LIN {X 0,Y 625.989,Z 663.19,A -85,B 0,C 180,E1 6456.402,E2 6456.402} C_VEL
LIN {X 0,Y 626.113,Z 663.19,A -85,B 0,C 180,E1 6463.797,E2 6463.797} C_VEL
LIN {X 0,Y 626.332,Z 663.19,A -85,B 0,C 180,E1 6470.922,E2 6470.922} C_VEL
LIN {X 0,Y 626.466,Z 663.19,A -85,B 0,C 180,E1 6477.902,E2 6477.902} C_VEL
LIN {X 0,Y 626.549,Z 663.19,A -85,B 0,C 180,E1 6484.849,E2 6484.849} C_VEL
LIN {X 0,Y 626.308,Z 663.19,A -85,B 0,C 180,E1 6493.295,E2 6493.295} C_VEL
LIN {X 0,Y 626.36,Z 663.19,A -85,B 0,C 180,E1 6501.237,E2 6501.237} C_VEL
LIN {X 0,Y 626.317,Z 663.19,A -85,B 0,C 180,E1 6509.77,E2 6509.77} C_VEL
LIN {X 0,Y 626.419,Z 663.19,A -85,B 0,C 180,E1 6518.14,E2 6518.14} C_VEL
LIN {X 0,Y 626.399,Z 664.346,A -85,B 0,C 180,E1 6525.792,E2 6525.792} C_VEL
LIN {X 0,Y 651.869,Z 715.355,A -85,B 0,C 180,E1 6528.472,E2 6528.472} C_VEL
LIN {X 0,Y 648.177,Z 791.571,A -85,B 0,C 180,E1 6530.446,E2 6530.446} C_VEL
LIN {X 0,Y 642.47,Z 861.614,A -85,B 0,C 180,E1 6533.738,E2 6533.738} C_VEL
LIN {X 0,Y 636.508,Z 924.999,A -85,B 0,C 180,E1 6538.337,E2 6538.337} C_VEL
LIN {X 0,Y 631.672,Z 978.511,A -85,B 0,C 180,E1 6544.011,E2 6544.011} C_VEL
LIN {X 0,Y 628.979,Z 1020.004,A -85,B 0,C 180,E1 6550.536,E2 6550.536} C_VEL
LIN {X 0,Y 627.568,Z 1047.097,A -85,B 0,C 180,E1 6557.439,E2 6557.439} C_VEL
LIN {X 0,Y 626.974,Z 1058.972,A -85,B 0,C 180,E1 6563.751,E2 6563.751} C_VEL
LIN {X 0,Y 627.176,Z 1059.603,A -85,B 0,C 180,E1 6569.307,E2 6569.307} C_VEL
LIN {X 0,Y 627.134,Z 1049.647,A -85,B 0,C 180,E1 6575.55,E2 6575.55} C_VEL
LIN {X 0,Y 627.887,Z 1027.464,A -85,B 0,C 180,E1 6581.846,E2 6581.846} C_VEL
LIN {X 0,Y 629.7,Z 1006.621,A -85,B 0,C 180,E1 6585.788,E2 6585.788} C_VEL
LIN {X 0,Y 622.562,Z 990.323,A -85,B 0,C 180,E1 6588.601,E2 6588.601} C_VEL
LIN {X 0,Y 627.357,Z 940.981,A -85,B 0,C 180,E1 6594.452,E2 6594.452} C_VEL
LIN {X 0,Y 633.854,Z 879.366,A -85,B 0,C 180,E1 6599.458,E2 6599.458} C_VEL
LIN {X 0,Y 640.199,Z 811.845,A -85,B 0,C 180,E1 6603.087,E2 6603.087} C_VEL
LIN {X 0,Y 644.763,Z 741.705,A -85,B 0,C 180,E1 6605.351,E2 6605.351} C_VEL
LIN {X 0,Y 644.279,Z 712.829,A -85,B 0,C 180,E1 6606.02,E2 6606.02} C_VEL
LIN {X 0,Y 618.028,Z 663.19,A -85,B 0,C 180,E1 6608.956,E2 6608.956} C_VEL
LIN {X 0,Y 618.105,Z 663.19,A -85,B 0,C 180,E1 6617.545,E2 6617.545} C_VEL
LIN {X 0,Y 618.102,Z 663.19,A -85,B 0,C 180,E1 6626.48,E2 6626.48} C_VEL
LIN {X 0,Y 618.278,Z 663.19,A -85,B 0,C 180,E1 6634.575,E2 6634.575} C_VEL
LIN {X 0,Y 618.593,Z 663.19,A -85,B 0,C 180,E1 6643.626,E2 6643.626} C_VEL
LIN {X 0,Y 618.803,Z 663.19,A -85,B 0,C 180,E1 6650.842,E2 6650.842} C_VEL
LIN {X 0,Y 619.166,Z 663.19,A -85,B 0,C 180,E1 6657.908,E2 6657.908} C_VEL
LIN {X 0,Y 618.585,Z 663.19,A -85,B 0,C 180,E1 6666.87,E2 6666.87} C_VEL
LIN {X 0,Y 618.331,Z 663.19,A -85,B 0,C 180,E1 6674.952,E2 6674.952} C_VEL
LIN {X 0,Y 618.059,Z 663.19,A -85,B 0,C 180,E1 6683.065,E2 6683.065} C_VEL
LIN {X 0,Y 618.548,Z 663.19,A -85,B 0,C 180,E1 6691.859,E2 6691.859} C_VEL
LIN {X 0,Y 618.263,Z 663.19,A -85,B 0,C 180,E1 6700.603,E2 6700.603} C_VEL
LIN {X 0,Y 618.318,Z 665.155,A -85,B 0,C 180,E1 6708.054,E2 6708.054} C_VEL
LIN {X 0,Y 645.805,Z 718.768,A -85,B 0,C 180,E1 6710.981,E2 6710.981} C_VEL
LIN {X 0,Y 642.302,Z 793.069,A -85,B 0,C 180,E1 6712.772,E2 6712.772} C_VEL
LIN {X 0,Y 636.489,Z 863.014,A -85,B 0,C 180,E1 6715.883,E2 6715.883} C_VEL
LIN {X 0,Y 630.05,Z 926.753,A -85,B 0,C 180,E1 6720.294,E2 6720.294} C_VEL
LIN {X 0,Y 624.493,Z 981.34,A -85,B 0,C 180,E1 6725.846,E2 6725.846} C_VEL
LIN {X 0,Y 621.095,Z 1024.089,A -85,B 0,C 180,E1 6732.231,E2 6732.231} C_VEL
LIN {X 0,Y 619.771,Z 1052.761,A -85,B 0,C 180,E1 6738.919,E2 6738.919} C_VEL
LIN {X 0,Y 619.545,Z 1067.017,A -85,B 0,C 180,E1 6745.086,E2 6745.086} C_VEL
LIN {X 0,Y 619.231,Z 1069.804,A -85,B 0,C 180,E1 6752.105,E2 6752.105} C_VEL
LIN {X 0,Y 619.104,Z 1060.28,A -85,B 0,C 180,E1 6758.451,E2 6758.451} C_VEL
LIN {X 0,Y 619.864,Z 1039.304,A -85,B 0,C 180,E1 6764.658,E2 6764.658} C_VEL
LIN {X 0,Y 622.106,Z 1006.633,A -85,B 0,C 180,E1 6770.698,E2 6770.698} C_VEL
LIN {X 0,Y 626.721,Z 958.006,A -85,B 0,C 180,E1 6776.784,E2 6776.784} C_VEL
LIN {X 0,Y 632.897,Z 898.514,A -85,B 0,C 180,E1 6781.89,E2 6781.89} C_VEL
LIN {X 0,Y 639.339,Z 831.694,A -85,B 0,C 180,E1 6785.706,E2 6785.706} C_VEL
LIN {X 0,Y 644.355,Z 760.024,A -85,B 0,C 180,E1 6788.194,E2 6788.194} C_VEL
LIN {X 0,Y 644.727,Z 712.454,A -85,B 0,C 180,E1 6789.202,E2 6789.202} C_VEL
LIN {X 0,Y 617.986,Z 663.19,A -85,B 0,C 180,E1 6792.181,E2 6792.181} C_VEL
LIN {X 0,Y 617.872,Z 663.19,A -85,B 0,C 180,E1 6801.195,E2 6801.195} C_VEL
LIN {X 0,Y 618.195,Z 663.19,A -85,B 0,C 180,E1 6809.763,E2 6809.763} C_VEL
LIN {X 0,Y 618.409,Z 663.19,A -85,B 0,C 180,E1 6819.136,E2 6819.136} C_VEL
LIN {X 0,Y 618.785,Z 663.19,A -85,B 0,C 180,E1 6827.95,E2 6827.95} C_VEL
LIN {X 0,Y 618.905,Z 663.19,A -85,B 0,C 180,E1 6836.47,E2 6836.47} C_VEL
LIN {X 0,Y 618.526,Z 663.19,A -85,B 0,C 180,E1 6844.912,E2 6844.912} C_VEL
LIN {X 0,Y 618.606,Z 663.19,A -85,B 0,C 180,E1 6852.022,E2 6852.022} C_VEL
LIN {X 0,Y 618.434,Z 663.19,A -85,B 0,C 180,E1 6860.83,E2 6860.83} C_VEL
LIN {X 0,Y 618.309,Z 663.19,A -85,B 0,C 180,E1 6869.466,E2 6869.466} C_VEL
LIN {X 0,Y 618.325,Z 663.19,A -85,B 0,C 180,E1 6877.15,E2 6877.15} C_VEL
LIN {X 0,Y 618.439,Z 665.18,A -85,B 0,C 180,E1 6885.154,E2 6885.154} C_VEL
LIN {X 0,Y 645.566,Z 717.694,A -85,B 0,C 180,E1 6888.064,E2 6888.064} C_VEL
LIN {X 0,Y 641.566,Z 793.048,A -85,B 0,C 180,E1 6890.072,E2 6890.072} C_VEL
LIN {X 0,Y 635.518,Z 862.685,A -85,B 0,C 180,E1 6893.399,E2 6893.399} C_VEL
LIN {X 0,Y 629.093,Z 926.353,A -85,B 0,C 180,E1 6898.095,E2 6898.095} C_VEL
LIN {X 0,Y 623.955,Z 979.19,A -85,B 0,C 180,E1 6903.799,E2 6903.799} C_VEL
LIN {X 0,Y 621.072,Z 1020.648,A -85,B 0,C 180,E1 6910.454,E2 6910.454} C_VEL
LIN {X 0,Y 619.649,Z 1046.987,A -85,B 0,C 180,E1 6917.276,E2 6917.276} C_VEL
LIN {X 0,Y 618.987,Z 1058.942,A -85,B 0,C 180,E1 6923.67,E2 6923.67} C_VEL
LIN {X 0,Y 619.176,Z 1059.632,A -85,B 0,C 180,E1 6929.298,E2 6929.298} C_VEL
LIN {X 0,Y 619.146,Z 1049.756,A -85,B 0,C 180,E1 6935.622,E2 6935.622} C_VEL
LIN {X 0,Y 619.919,Z 1029.339,A -85,B 0,C 180,E1 6941.604,E2 6941.604} C_VEL
LIN {X 0,Y 622.168,Z 996.079,A -85,B 0,C 180,E1 6947.738,E2 6947.738} C_VEL
LIN {X 0,Y 622.562,Z 990.323,A -85,B 0,C 180,E1 6948.601,E2 6948.601} C_VEL
LIN {X 0,Y 617.22,Z 971.758,A -85,B 0,C 180,E1 6951.357,E2 6951.357} C_VEL
LIN {X 0,Y 622.951,Z 916.676,A -85,B 0,C 180,E1 6957.041,E2 6957.041} C_VEL
LIN {X 0,Y 629.604,Z 853.137,A -85,B 0,C 180,E1 6961.489,E2 6961.489} C_VEL
LIN {X 0,Y 635.961,Z 781.489,A -85,B 0,C 180,E1 6964.683,E2 6964.683} C_VEL
LIN {X 0,Y 638.105,Z 715.966,A -85,B 0,C 180,E1 6966.419,E2 6966.419} C_VEL
LIN {X 0,Y 609.903,Z 663.19,A -85,B 0,C 180,E1 6969.693,E2 6969.693} C_VEL
LIN {X 0,Y 610.126,Z 663.19,A -85,B 0,C 180,E1 6977.154,E2 6977.154} C_VEL
LIN {X 0,Y 610.092,Z 663.19,A -85,B 0,C 180,E1 6986.372,E2 6986.372} C_VEL
LIN {X 0,Y 610.278,Z 663.19,A -85,B 0,C 180,E1 6995.086,E2 6995.086} C_VEL
LIN {X 0,Y 610.527,Z 663.19,A -85,B 0,C 180,E1 7003.404,E2 7003.404} C_VEL
LIN {X 0,Y 610.82,Z 663.19,A -85,B 0,C 180,E1 7010.721,E2 7010.721} C_VEL
LIN {X 0,Y 611.183,Z 663.19,A -85,B 0,C 180,E1 7017.881,E2 7017.881} C_VEL
LIN {X 0,Y 610.717,Z 663.19,A -85,B 0,C 180,E1 7026.437,E2 7026.437} C_VEL
LIN {X 0,Y 610.275,Z 663.19,A -85,B 0,C 180,E1 7035.154,E2 7035.154} C_VEL
LIN {X 0,Y 610.13,Z 663.19,A -85,B 0,C 180,E1 7042.697,E2 7042.697} C_VEL
LIN {X 0,Y 610.501,Z 663.19,A -85,B 0,C 180,E1 7051.026,E2 7051.026} C_VEL
LIN {X 0,Y 610.256,Z 663.19,A -85,B 0,C 180,E1 7059.382,E2 7059.382} C_VEL
LIN {X 0,Y 610.188,Z 664.755,A -85,B 0,C 180,E1 7067.37,E2 7067.37} C_VEL
LIN {X 0,Y 639.531,Z 721.3,A -85,B 0,C 180,E1 7070.569,E2 7070.569} C_VEL
LIN {X 0,Y 635.739,Z 794.861,A -85,B 0,C 180,E1 7072.394,E2 7072.394} C_VEL
LIN {X 0,Y 629.598,Z 864.163,A -85,B 0,C 180,E1 7075.528,E2 7075.528} C_VEL
LIN {X 0,Y 622.672,Z 928.343,A -85,B 0,C 180,E1 7080.05,E2 7080.05} C_VEL
LIN {X 0,Y 616.761,Z 982.879,A -85,B 0,C 180,E1 7085.726,E2 7085.726} C_VEL
LIN {X 0,Y 613.197,Z 1025.473,A -85,B 0,C 180,E1 7092.258,E2 7092.258} C_VEL
LIN {X 0,Y 611.857,Z 1054.394,A -85,B 0,C 180,E1 7099.288,E2 7099.288} C_VEL
LIN {X 0,Y 611.057,Z 1068.735,A -85,B 0,C 180,E1 7106.443,E2 7106.443} C_VEL
LIN {X 0,Y 611.217,Z 1069.804,A -85,B 0,C 180,E1 7112.133,E2 7112.133} C_VEL
LIN {X 0,Y 611.106,Z 1060.28,A -85,B 0,C 180,E1 7118.563,E2 7118.563} C_VEL
LIN {X 0,Y 611.921,Z 1039.774,A -85,B 0,C 180,E1 7124.74,E2 7124.74} C_VEL
LIN {X 0,Y 614.345,Z 1006.631,A -85,B 0,C 180,E1 7130.972,E2 7130.972} C_VEL
LIN {X 0,Y 619.276,Z 958.172,A -85,B 0,C 180,E1 7137.113,E2 7137.113} C_VEL
LIN {X 0,Y 625.962,Z 898.034,A -85,B 0,C 180,E1 7142.322,E2 7142.322} C_VEL
LIN {X 0,Y 632.78,Z 831.525,A -85,B 0,C 180,E1 7146.141,E2 7146.141} C_VEL
LIN {X 0,Y 638.057,Z 759.411,A -85,B 0,C 180,E1 7148.655,E2 7148.655} C_VEL
LIN {X 0,Y 638.305,Z 715.18,A -85,B 0,C 180,E1 7149.625,E2 7149.625} C_VEL
LIN {X 0,Y 610.038,Z 663.19,A -85,B 0,C 180,E1 7152.757,E2 7152.757} C_VEL
LIN {X 0,Y 609.871,Z 663.19,A -85,B 0,C 180,E1 7161.558,E2 7161.558} C_VEL
LIN {X 0,Y 610.255,Z 663.19,A -85,B 0,C 180,E1 7170.97,E2 7170.97} C_VEL
LIN {X 0,Y 610.396,Z 663.19,A -85,B 0,C 180,E1 7180.369,E2 7180.369} C_VEL
LIN {X 0,Y 610.575,Z 663.19,A -85,B 0,C 180,E1 7189.239,E2 7189.239} C_VEL
LIN {X 0,Y 610.917,Z 663.19,A -85,B 0,C 180,E1 7196.424,E2 7196.424} C_VEL
LIN {X 0,Y 611.171,Z 663.19,A -85,B 0,C 180,E1 7203.544,E2 7203.544} C_VEL
LIN {X 0,Y 610.553,Z 663.19,A -85,B 0,C 180,E1 7212.183,E2 7212.183} C_VEL
LIN {X 0,Y 610.375,Z 663.19,A -85,B 0,C 180,E1 7221.118,E2 7221.118} C_VEL
LIN {X 0,Y 610.299,Z 663.19,A -85,B 0,C 180,E1 7228.992,E2 7228.992} C_VEL
LIN {X 0,Y 610.296,Z 663.19,A -85,B 0,C 180,E1 7237.52,E2 7237.52} C_VEL
LIN {X 0,Y 610.298,Z 665.046,A -85,B 0,C 180,E1 7244.451,E2 7244.451} C_VEL
LIN {X 0,Y 639.271,Z 719.493,A -85,B 0,C 180,E1 7247.644,E2 7247.644} C_VEL
LIN {X 0,Y 634.992,Z 794.438,A -85,B 0,C 180,E1 7249.684,E2 7249.684} C_VEL
LIN {X 0,Y 628.464,Z 864.635,A -85,B 0,C 180,E1 7253.103,E2 7253.103} C_VEL
LIN {X 0,Y 621.74,Z 927.168,A -85,B 0,C 180,E1 7257.798,E2 7257.798} C_VEL
LIN {X 0,Y 616.267,Z 979.509,A -85,B 0,C 180,E1 7263.535,E2 7263.535} C_VEL
LIN {X 0,Y 613.144,Z 1020.442,A -85,B 0,C 180,E1 7270.191,E2 7270.191} C_VEL
LIN {X 0,Y 611.714,Z 1046.878,A -85,B 0,C 180,E1 7277.108,E2 7277.108} C_VEL
LIN {X 0,Y 611.011,Z 1058.913,A -85,B 0,C 180,E1 7283.587,E2 7283.587} C_VEL
LIN {X 0,Y 611.197,Z 1059.66,A -85,B 0,C 180,E1 7289.289,E2 7289.289} C_VEL
LIN {X 0,Y 611.148,Z 1049.864,A -85,B 0,C 180,E1 7295.696,E2 7295.696} C_VEL
LIN {X 0,Y 611.978,Z 1029.194,A -85,B 0,C 180,E1 7301.832,E2 7301.832} C_VEL
LIN {X 0,Y 614.41,Z 995.857,A -85,B 0,C 180,E1 7308.047,E2 7308.047} C_VEL
LIN {X 0,Y 617.22,Z 971.758,A -85,B 0,C 180,E1 7311.357,E2 7311.357} C_VEL
LIN {X 0,Y 611.43,Z 951.715,A -85,B 0,C 180,E1 7314.042,E2 7314.042} C_VEL
LIN {X 0,Y 618.594,Z 892.06,A -85,B 0,C 180,E1 7319.381,E2 7319.381} C_VEL
LIN {X 0,Y 625.879,Z 825.182,A -85,B 0,C 180,E1 7323.375,E2 7323.375} C_VEL
LIN {X 0,Y 631.561,Z 752.877,A -85,B 0,C 180,E1 7325.996,E2 7325.996} C_VEL
LIN {X 0,Y 631.694,Z 718.464,A -85,B 0,C 180,E1 7326.856,E2 7326.856} C_VEL
LIN {X 0,Y 601.853,Z 663.19,A -85,B 0,C 180,E1 7330.342,E2 7330.342} C_VEL
LIN {X 0,Y 602,Z 663.19,A -85,B 0,C 180,E1 7338.098,E2 7338.098} C_VEL
LIN {X 0,Y 602.138,Z 663.19,A -85,B 0,C 180,E1 7347.203,E2 7347.203} C_VEL
LIN {X 0,Y 602.32,Z 663.19,A -85,B 0,C 180,E1 7355.449,E2 7355.449} C_VEL
LIN {X 0,Y 602.823,Z 663.19,A -85,B 0,C 180,E1 7364.687,E2 7364.687} C_VEL
LIN {X 0,Y 602.465,Z 663.19,A -85,B 0,C 180,E1 7372.051,E2 7372.051} C_VEL
LIN {X 0,Y 602.554,Z 663.19,A -85,B 0,C 180,E1 7379.294,E2 7379.294} C_VEL
LIN {X 0,Y 602.709,Z 663.19,A -85,B 0,C 180,E1 7386.523,E2 7386.523} C_VEL
LIN {X 0,Y 602.233,Z 663.19,A -85,B 0,C 180,E1 7395.361,E2 7395.361} C_VEL
LIN {X 0,Y 602.022,Z 663.19,A -85,B 0,C 180,E1 7403.164,E2 7403.164} C_VEL
LIN {X 0,Y 602.505,Z 663.19,A -85,B 0,C 180,E1 7411.111,E2 7411.111} C_VEL
LIN {X 0,Y 602.233,Z 663.19,A -85,B 0,C 180,E1 7420.011,E2 7420.011} C_VEL
LIN {X 0,Y 602.125,Z 664.619,A -85,B 0,C 180,E1 7426.675,E2 7426.675} C_VEL
LIN {X 0,Y 633.316,Z 722.987,A -85,B 0,C 180,E1 7430.135,E2 7430.135} C_VEL
LIN {X 0,Y 629.168,Z 797.343,A -85,B 0,C 180,E1 7432.031,E2 7432.031} C_VEL
LIN {X 0,Y 622.501,Z 867.6,A -85,B 0,C 180,E1 7435.297,E2 7435.297} C_VEL
LIN {X 0,Y 615.215,Z 930.645,A -85,B 0,C 180,E1 7439.873,E2 7439.873} C_VEL
LIN {X 0,Y 608.925,Z 985.452,A -85,B 0,C 180,E1 7445.739,E2 7445.739} C_VEL
LIN {X 0,Y 605.274,Z 1026.854,A -85,B 0,C 180,E1 7452.285,E2 7452.285} C_VEL
LIN {X 0,Y 603.907,Z 1055.519,A -85,B 0,C 180,E1 7459.511,E2 7459.511} C_VEL
LIN {X 0,Y 603.066,Z 1068.735,A -85,B 0,C 180,E1 7466.396,E2 7466.396} C_VEL
LIN {X 0,Y 603.205,Z 1069.805,A -85,B 0,C 180,E1 7472.161,E2 7472.161} C_VEL
LIN {X 0,Y 603.127,Z 1060.281,A -85,B 0,C 180,E1 7478.677,E2 7478.677} C_VEL
LIN {X 0,Y 603.972,Z 1040.223,A -85,B 0,C 180,E1 7484.829,E2 7484.829} C_VEL
LIN {X 0,Y 606.511,Z 1007.671,A -85,B 0,C 180,E1 7491.09,E2 7491.09} C_VEL
LIN {X 0,Y 611.714,Z 959.739,A -85,B 0,C 180,E1 7497.298,E2 7497.298} C_VEL
LIN {X 0,Y 618.824,Z 899.5,A -85,B 0,C 180,E1 7502.624,E2 7502.624} C_VEL
LIN {X 0,Y 626.099,Z 832.698,A -85,B 0,C 180,E1 7506.525,E2 7506.525} C_VEL
LIN {X 0,Y 631.688,Z 760.974,A -85,B 0,C 180,E1 7509.072,E2 7509.072} C_VEL
LIN {X 0,Y 632.081,Z 718.258,A -85,B 0,C 180,E1 7510.039,E2 7510.039} C_VEL
LIN {X 0,Y 602.03,Z 663.19,A -85,B 0,C 180,E1 7513.5,E2 7513.5} C_VEL
LIN {X 0,Y 601.938,Z 663.19,A -85,B 0,C 180,E1 7522.519,E2 7522.519} C_VEL
LIN {X 0,Y 602.161,Z 663.19,A -85,B 0,C 180,E1 7530.542,E2 7530.542} C_VEL
LIN {X 0,Y 602.36,Z 663.19,A -85,B 0,C 180,E1 7540.097,E2 7540.097} C_VEL
LIN {X 0,Y 602.585,Z 663.19,A -85,B 0,C 180,E1 7549.095,E2 7549.095} C_VEL
LIN {X 0,Y 602.92,Z 663.19,A -85,B 0,C 180,E1 7556.376,E2 7556.376} C_VEL
LIN {X 0,Y 603.132,Z 663.19,A -85,B 0,C 180,E1 7563.591,E2 7563.591} C_VEL
LIN {X 0,Y 602.496,Z 663.19,A -85,B 0,C 180,E1 7572.348,E2 7572.348} C_VEL
LIN {X 0,Y 602.345,Z 663.19,A -85,B 0,C 180,E1 7581.414,E2 7581.414} C_VEL
LIN {X 0,Y 602.251,Z 663.19,A -85,B 0,C 180,E1 7589.694,E2 7589.694} C_VEL
LIN {X 0,Y 602.283,Z 663.19,A -85,B 0,C 180,E1 7598.108,E2 7598.108} C_VEL
LIN {X 0,Y 602.263,Z 665.134,A -85,B 0,C 180,E1 7603.728,E2 7603.728} C_VEL
LIN {X 0,Y 632.957,Z 722.137,A -85,B 0,C 180,E1 7607.233,E2 7607.233} C_VEL
LIN {X 0,Y 628.153,Z 798.434,A -85,B 0,C 180,E1 7609.384,E2 7609.384} C_VEL
LIN {X 0,Y 621.227,Z 868.652,A -85,B 0,C 180,E1 7612.93,E2 7612.93} C_VEL
LIN {X 0,Y 614.205,Z 930.063,A -85,B 0,C 180,E1 7617.685,E2 7617.685} C_VEL
LIN {X 0,Y 608.374,Z 982.733,A -85,B 0,C 180,E1 7623.67,E2 7623.67} C_VEL
LIN {X 0,Y 605.22,Z 1021.68,A -85,B 0,C 180,E1 7630.229,E2 7630.229} C_VEL
LIN {X 0,Y 603.785,Z 1046.768,A -85,B 0,C 180,E1 7636.936,E2 7636.936} C_VEL
LIN {X 0,Y 602.999,Z 1059.027,A -85,B 0,C 180,E1 7643.702,E2 7643.702} C_VEL
LIN {X 0,Y 603.196,Z 1059.689,A -85,B 0,C 180,E1 7649.279,E2 7649.279} C_VEL
LIN {X 0,Y 603.162,Z 1050.094,A -85,B 0,C 180,E1 7655.718,E2 7655.718} C_VEL
LIN {X 0,Y 604.04,Z 1029.061,A -85,B 0,C 180,E1 7662.065,E2 7662.065} C_VEL
LIN {X 0,Y 606.693,Z 995.443,A -85,B 0,C 180,E1 7668.394,E2 7668.394} C_VEL
LIN {X 0,Y 611.43,Z 951.715,A -85,B 0,C 180,E1 7674.042,E2 7674.042} C_VEL
LIN {X 0,Y 606.879,Z 929.837,A -85,B 0,C 180,E1 7676.636,E2 7676.636} C_VEL
LIN {X 0,Y 614.715,Z 866.262,A -85,B 0,C 180,E1 7681.561,E2 7681.561} C_VEL
LIN {X 0,Y 621.985,Z 797.253,A -85,B 0,C 180,E1 7685.021,E2 7685.021} C_VEL
LIN {X 0,Y 626.889,Z 727.794,A -85,B 0,C 180,E1 7687.011,E2 7687.011} C_VEL
LIN {X 0,Y 602.756,Z 679.837,A -85,B 0,C 180,E1 7689.849,E2 7689.849} C_VEL
LIN {X 0,Y 593.856,Z 663.19,A -85,B 0,C 180,E1 7691.089,E2 7691.089} C_VEL
LIN {X 0,Y 593.937,Z 663.19,A -85,B 0,C 180,E1 7699.355,E2 7699.355} C_VEL
LIN {X 0,Y 594.246,Z 663.19,A -85,B 0,C 180,E1 7708.744,E2 7708.744} C_VEL
LIN {X 0,Y 594.424,Z 663.19,A -85,B 0,C 180,E1 7718.287,E2 7718.287} C_VEL
LIN {X 0,Y 595.208,Z 663.19,A -85,B 0,C 180,E1 7727.498,E2 7727.498} C_VEL
LIN {X 0,Y 595.176,Z 663.19,A -85,B 0,C 180,E1 7737.824,E2 7737.824} C_VEL
LIN {X 0,Y 594.672,Z 663.19,A -85,B 0,C 180,E1 7746.611,E2 7746.611} C_VEL
LIN {X 0,Y 594.189,Z 663.19,A -85,B 0,C 180,E1 7755.574,E2 7755.574} C_VEL
LIN {X 0,Y 593.997,Z 663.19,A -85,B 0,C 180,E1 7763.349,E2 7763.349} C_VEL
LIN {X 0,Y 594.505,Z 663.19,A -85,B 0,C 180,E1 7771.577,E2 7771.577} C_VEL
LIN {X 0,Y 594.145,Z 663.19,A -85,B 0,C 180,E1 7780.669,E2 7780.669} C_VEL
LIN {X 0,Y 594.206,Z 665.179,A -85,B 0,C 180,E1 7785.982,E2 7785.982} C_VEL
LIN {X 0,Y 627.136,Z 724.807,A -85,B 0,C 180,E1 7789.696,E2 7789.696} C_VEL
LIN {X 0,Y 622.711,Z 798.447,A -85,B 0,C 180,E1 7791.613,E2 7791.613} C_VEL
LIN {X 0,Y 615.771,Z 867.404,A -85,B 0,C 180,E1 7794.855,E2 7794.855} C_VEL
LIN {X 0,Y 607.996,Z 930.747,A -85,B 0,C 180,E1 7799.488,E2 7799.488} C_VEL
LIN {X 0,Y 601.331,Z 985.45,A -85,B 0,C 180,E1 7805.412,E2 7805.412} C_VEL
LIN {X 0,Y 597.417,Z 1026.619,A -85,B 0,C 180,E1 7811.999,E2 7811.999} C_VEL
LIN {X 0,Y 595.916,Z 1055.519,A -85,B 0,C 180,E1 7819.369,E2 7819.369} C_VEL
LIN {X 0,Y 595.075,Z 1068.735,A -85,B 0,C 180,E1 7826.348,E2 7826.348} C_VEL
LIN {X 0,Y 595.196,Z 1069.805,A -85,B 0,C 180,E1 7832.191,E2 7832.191} C_VEL
LIN {X 0,Y 595.157,Z 1060.281,A -85,B 0,C 180,E1 7838.794,E2 7838.794} C_VEL
LIN {X 0,Y 596.069,Z 1039.801,A -85,B 0,C 180,E1 7845.134,E2 7845.134} C_VEL
LIN {X 0,Y 598.837,Z 1006.627,A -85,B 0,C 180,E1 7851.542,E2 7851.542} C_VEL
LIN {X 0,Y 604.492,Z 958.579,A -85,B 0,C 180,E1 7857.785,E2 7857.785} C_VEL
LIN {X 0,Y 612.042,Z 898.208,A -85,B 0,C 180,E1 7863.136,E2 7863.136} C_VEL
LIN {X 0,Y 619.721,Z 830.554,A -85,B 0,C 180,E1 7867.068,E2 7867.068} C_VEL
LIN {X 0,Y 625.488,Z 760.438,A -85,B 0,C 180,E1 7869.547,E2 7869.547} C_VEL
LIN {X 0,Y 626.028,Z 721.828,A -85,B 0,C 180,E1 7870.442,E2 7870.442} C_VEL
LIN {X 0,Y 593.995,Z 663.19,A -85,B 0,C 180,E1 7874.303,E2 7874.303} C_VEL
LIN {X 0,Y 593.987,Z 663.19,A -85,B 0,C 180,E1 7883.531,E2 7883.531} C_VEL
LIN {X 0,Y 594.137,Z 663.19,A -85,B 0,C 180,E1 7891.779,E2 7891.779} C_VEL
LIN {X 0,Y 594.26,Z 663.19,A -85,B 0,C 180,E1 7901.365,E2 7901.365} C_VEL
LIN {X 0,Y 594.597,Z 663.19,A -85,B 0,C 180,E1 7909.076,E2 7909.076} C_VEL
LIN {X 0,Y 594.943,Z 663.19,A -85,B 0,C 180,E1 7916.327,E2 7916.327} C_VEL
LIN {X 0,Y 595.103,Z 663.19,A -85,B 0,C 180,E1 7923.64,E2 7923.64} C_VEL
LIN {X 0,Y 594.462,Z 663.19,A -85,B 0,C 180,E1 7932.518,E2 7932.518} C_VEL
LIN {X 0,Y 594.345,Z 663.19,A -85,B 0,C 180,E1 7941.367,E2 7941.367} C_VEL
LIN {X 0,Y 594.27,Z 663.19,A -85,B 0,C 180,E1 7949.852,E2 7949.852} C_VEL
LIN {X 0,Y 594.196,Z 663.19,A -85,B 0,C 180,E1 7958.888,E2 7958.888} C_VEL
LIN {X 0,Y 594.178,Z 664.681,A -85,B 0,C 180,E1 7962.959,E2 7962.959} C_VEL
LIN {X 0,Y 626.665,Z 725.464,A -85,B 0,C 180,E1 7966.828,E2 7966.828} C_VEL
LIN {X 0,Y 621.473,Z 801.297,A -85,B 0,C 180,E1 7969.036,E2 7969.036} C_VEL
LIN {X 0,Y 614.251,Z 870.321,A -85,B 0,C 180,E1 7972.602,E2 7972.602} C_VEL
LIN {X 0,Y 606.738,Z 932.12,A -85,B 0,C 180,E1 7977.496,E2 7977.496} C_VEL
LIN {X 0,Y 600.591,Z 984.389,A -85,B 0,C 180,E1 7983.596,E2 7983.596} C_VEL
LIN {X 0,Y 597.242,Z 1023.242,A -85,B 0,C 180,E1 7990.341,E2 7990.341} C_VEL
LIN {X 0,Y 595.563,Z 1048.603,A -85,B 0,C 180,E1 7997.5,E2 7997.5} C_VEL
LIN {X 0,Y 595.035,Z 1058.852,A -85,B 0,C 180,E1 8003.414,E2 8003.414} C_VEL
LIN {X 0,Y 595.196,Z 1059.718,A -85,B 0,C 180,E1 8009.27,E2 8009.27} C_VEL
LIN {X 0,Y 595.187,Z 1050.422,A -85,B 0,C 180,E1 8015.682,E2 8015.682} C_VEL
LIN {X 0,Y 596.127,Z 1029.377,A -85,B 0,C 180,E1 8022.192,E2 8022.192} C_VEL
LIN {X 0,Y 598.858,Z 996.901,A -85,B 0,C 180,E1 8028.452,E2 8028.452} C_VEL
LIN {X 0,Y 604.224,Z 949.905,A -85,B 0,C 180,E1 8034.6,E2 8034.6} C_VEL
LIN {X 0,Y 606.879,Z 929.837,A -85,B 0,C 180,E1 8036.636,E2 8036.636} C_VEL
LIN {X 0,Y 602.959,Z 906.153,A -85,B 0,C 180,E1 8039.116,E2 8039.116} C_VEL
LIN {X 0,Y 610.993,Z 841.438,A -85,B 0,C 180,E1 8043.466,E2 8043.466} C_VEL
LIN {X 0,Y 617.769,Z 769.522,A -85,B 0,C 180,E1 8046.476,E2 8046.476} C_VEL
LIN {X 0,Y 619.37,Z 724.87,A -85,B 0,C 180,E1 8047.668,E2 8047.668} C_VEL
LIN {X 0,Y 585.806,Z 663.19,A -85,B 0,C 180,E1 8051.721,E2 8051.721} C_VEL
LIN {X 0,Y 585.939,Z 663.19,A -85,B 0,C 180,E1 8060.628,E2 8060.628} C_VEL
LIN {X 0,Y 586.265,Z 663.19,A -85,B 0,C 180,E1 8070.054,E2 8070.054} C_VEL
LIN {X 0,Y 586.322,Z 663.19,A -85,B 0,C 180,E1 8079.562,E2 8079.562} C_VEL
LIN {X 0,Y 587.204,Z 663.19,A -85,B 0,C 180,E1 8088.838,E2 8088.838} C_VEL
LIN {X 0,Y 587.171,Z 663.19,A -85,B 0,C 180,E1 8097.794,E2 8097.794} C_VEL
LIN {X 0,Y 586.64,Z 663.19,A -85,B 0,C 180,E1 8106.702,E2 8106.702} C_VEL
LIN {X 0,Y 586.426,Z 663.19,A -85,B 0,C 180,E1 8114.25,E2 8114.25} C_VEL
LIN {X 0,Y 586.014,Z 663.19,A -85,B 0,C 180,E1 8123.275,E2 8123.275} C_VEL
LIN {X 0,Y 586.435,Z 663.19,A -85,B 0,C 180,E1 8132.063,E2 8132.063} C_VEL
LIN {X 0,Y 586.144,Z 663.19,A -85,B 0,C 180,E1 8141.345,E2 8141.345} C_VEL
LIN {X 0,Y 586.043,Z 664.442,A -85,B 0,C 180,E1 8145.22,E2 8145.22} C_VEL
LIN {X 0,Y 620.93,Z 728.091,A -85,B 0,C 180,E1 8149.271,E2 8149.271} C_VEL
LIN {X 0,Y 615.969,Z 802.174,A -85,B 0,C 180,E1 8151.284,E2 8151.284} C_VEL
LIN {X 0,Y 608.464,Z 871.966,A -85,B 0,C 180,E1 8154.699,E2 8154.699} C_VEL
LIN {X 0,Y 600.273,Z 935.635,A -85,B 0,C 180,E1 8159.541,E2 8159.541} C_VEL
LIN {X 0,Y 593.364,Z 989.126,A -85,B 0,C 180,E1 8165.567,E2 8165.567} C_VEL
LIN {X 0,Y 589.422,Z 1030.103,A -85,B 0,C 180,E1 8172.464,E2 8172.464} C_VEL
LIN {X 0,Y 587.9,Z 1056.487,A -85,B 0,C 180,E1 8179.598,E2 8179.598} C_VEL
LIN {X 0,Y 587.083,Z 1068.736,A -85,B 0,C 180,E1 8186.298,E2 8186.298} C_VEL
LIN {X 0,Y 587.183,Z 1069.805,A -85,B 0,C 180,E1 8192.22,E2 8192.22} C_VEL
LIN {X 0,Y 587.186,Z 1060.281,A -85,B 0,C 180,E1 8198.914,E2 8198.914} C_VEL
LIN {X 0,Y 588.18,Z 1039.685,A -85,B 0,C 180,E1 8205.371,E2 8205.371} C_VEL
LIN {X 0,Y 591.078,Z 1006.625,A -85,B 0,C 180,E1 8211.839,E2 8211.839} C_VEL
LIN {X 0,Y 597.002,Z 959.736,A -85,B 0,C 180,E1 8218.029,E2 8218.029} C_VEL
LIN {X 0,Y 604.773,Z 900.68,A -85,B 0,C 180,E1 8223.372,E2 8223.372} C_VEL
LIN {X 0,Y 612.911,Z 833.884,A -85,B 0,C 180,E1 8227.372,E2 8227.372} C_VEL
LIN {X 0,Y 619.167,Z 762.445,A -85,B 0,C 180,E1 8229.971,E2 8229.971} C_VEL
LIN {X 0,Y 619.738,Z 724.649,A -85,B 0,C 180,E1 8230.887,E2 8230.887} C_VEL
LIN {X 0,Y 585.947,Z 663.19,A -85,B 0,C 180,E1 8234.993,E2 8234.993} C_VEL
LIN {X 0,Y 585.933,Z 663.19,A -85,B 0,C 180,E1 8244.611,E2 8244.611} C_VEL
LIN {X 0,Y 586.033,Z 663.19,A -85,B 0,C 180,E1 8253.218,E2 8253.218} C_VEL
LIN {X 0,Y 586.239,Z 663.19,A -85,B 0,C 180,E1 8261.101,E2 8261.101} C_VEL
LIN {X 0,Y 586.584,Z 663.19,A -85,B 0,C 180,E1 8268.794,E2 8268.794} C_VEL
LIN {X 0,Y 586.944,Z 663.19,A -85,B 0,C 180,E1 8276.277,E2 8276.277} C_VEL
LIN {X 0,Y 587.065,Z 663.19,A -85,B 0,C 180,E1 8283.69,E2 8283.69} C_VEL
LIN {X 0,Y 586.414,Z 663.19,A -85,B 0,C 180,E1 8292.693,E2 8292.693} C_VEL
LIN {X 0,Y 586.402,Z 663.19,A -85,B 0,C 180,E1 8300.435,E2 8300.435} C_VEL
LIN {X 0,Y 586.269,Z 663.19,A -85,B 0,C 180,E1 8308.598,E2 8308.598} C_VEL
LIN {X 0,Y 586.176,Z 663.19,A -85,B 0,C 180,E1 8317.46,E2 8317.46} C_VEL
LIN {X 0,Y 586.273,Z 665.19,A -85,B 0,C 180,E1 8322.189,E2 8322.189} C_VEL
LIN {X 0,Y 620.455,Z 727.52,A -85,B 0,C 180,E1 8326.39,E2 8326.39} C_VEL
LIN {X 0,Y 614.991,Z 802.702,A -85,B 0,C 180,E1 8328.625,E2 8328.625} C_VEL
LIN {X 0,Y 607.267,Z 872.234,A -85,B 0,C 180,E1 8332.28,E2 8332.28} C_VEL
LIN {X 0,Y 599.346,Z 933.232,A -85,B 0,C 180,E1 8337.217,E2 8337.217} C_VEL
LIN {X 0,Y 592.867,Z 985.289,A -85,B 0,C 180,E1 8343.409,E2 8343.409} C_VEL
LIN {X 0,Y 589.287,Z 1024.175,A -85,B 0,C 180,E1 8350.316,E2 8350.316} C_VEL
LIN {X 0,Y 587.617,Z 1048.493,A -85,B 0,C 180,E1 8357.329,E2 8357.329} C_VEL
LIN {X 0,Y 587.042,Z 1058.814,A -85,B 0,C 180,E1 8363.324,E2 8363.324} C_VEL
LIN {X 0,Y 587.197,Z 1059.747,A -85,B 0,C 180,E1 8369.26,E2 8369.26} C_VEL
LIN {X 0,Y 587.173,Z 1049.847,A -85,B 0,C 180,E1 8376.062,E2 8376.062} C_VEL
LIN {X 0,Y 588.287,Z 1028.351,A -85,B 0,C 180,E1 8382.656,E2 8382.656} C_VEL
LIN {X 0,Y 591.358,Z 994.805,A -85,B 0,C 180,E1 8389.083,E2 8389.083} C_VEL
LIN {X 0,Y 597.408,Z 946.076,A -85,B 0,C 180,E1 8395.393,E2 8395.393} C_VEL
LIN {X 0,Y 602.959,Z 906.153,A -85,B 0,C 180,E1 8399.116,E2 8399.116} C_VEL
LIN {X 0,Y 599.358,Z 880.945,A -85,B 0,C 180,E1 8401.473,E2 8401.473} C_VEL
LIN {X 0,Y 607.71,Z 813.296,A -85,B 0,C 180,E1 8405.297,E2 8405.297} C_VEL
LIN {X 0,Y 613.659,Z 744.456,A -85,B 0,C 180,E1 8407.618,E2 8407.618} C_VEL
LIN {X 0,Y 612.752,Z 726.894,A -85,B 0,C 180,E1 8408.156,E2 8408.156} C_VEL
LIN {X 0,Y 577.85,Z 663.19,A -85,B 0,C 180,E1 8412.444,E2 8412.444} C_VEL
LIN {X 0,Y 577.931,Z 663.19,A -85,B 0,C 180,E1 8420.717,E2 8420.717} C_VEL
LIN {X 0,Y 578.161,Z 663.19,A -85,B 0,C 180,E1 8429.228,E2 8429.228} C_VEL
LIN {X 0,Y 578.328,Z 663.19,A -85,B 0,C 180,E1 8438.564,E2 8438.564} C_VEL
LIN {X 0,Y 579.122,Z 663.19,A -85,B 0,C 180,E1 8447.145,E2 8447.145} C_VEL
LIN {X 0,Y 579.177,Z 663.19,A -85,B 0,C 180,E1 8457.763,E2 8457.763} C_VEL
LIN {X 0,Y 578.606,Z 663.19,A -85,B 0,C 180,E1 8466.796,E2 8466.796} C_VEL
LIN {X 0,Y 578.365,Z 663.19,A -85,B 0,C 180,E1 8474.453,E2 8474.453} C_VEL
LIN {X 0,Y 578.077,Z 663.19,A -85,B 0,C 180,E1 8482.395,E2 8482.395} C_VEL
LIN {X 0,Y 578.4,Z 663.19,A -85,B 0,C 180,E1 8491.564,E2 8491.564} C_VEL
LIN {X 0,Y 578.122,Z 663.19,A -85,B 0,C 180,E1 8500.053,E2 8500.053} C_VEL
LIN {X 0,Y 578.113,Z 664.757,A -85,B 0,C 180,E1 8504.469,E2 8504.469} C_VEL
LIN {X 0,Y 614.624,Z 731.797,A -85,B 0,C 180,E1 8508.854,E2 8508.854} C_VEL
LIN {X 0,Y 609.282,Z 805.755,A -85,B 0,C 180,E1 8510.951,E2 8510.951} C_VEL
LIN {X 0,Y 601.364,Z 874.966,A -85,B 0,C 180,E1 8514.441,E2 8514.441} C_VEL
LIN {X 0,Y 592.823,Z 937.99,A -85,B 0,C 180,E1 8519.359,E2 8519.359} C_VEL
LIN {X 0,Y 585.6,Z 991.043,A -85,B 0,C 180,E1 8525.496,E2 8525.496} C_VEL
LIN {X 0,Y 581.487,Z 1031.584,A -85,B 0,C 180,E1 8532.549,E2 8532.549} C_VEL
LIN {X 0,Y 579.656,Z 1058.416,A -85,B 0,C 180,E1 8540.21,E2 8540.21} C_VEL
LIN {X 0,Y 579.117,Z 1068.736,A -85,B 0,C 180,E1 8546.247,E2 8546.247} C_VEL
LIN {X 0,Y 579.171,Z 1069.805,A -85,B 0,C 180,E1 8552.251,E2 8552.251} C_VEL
LIN {X 0,Y 579.187,Z 1060.281,A -85,B 0,C 180,E1 8559.038,E2 8559.038} C_VEL
LIN {X 0,Y 580.259,Z 1039.875,A -85,B 0,C 180,E1 8565.538,E2 8565.538} C_VEL
LIN {X 0,Y 583.41,Z 1006.623,A -85,B 0,C 180,E1 8572.141,E2 8572.141} C_VEL
LIN {X 0,Y 589.879,Z 958.229,A -85,B 0,C 180,E1 8578.577,E2 8578.577} C_VEL
LIN {X 0,Y 598.242,Z 898.302,A -85,B 0,C 180,E1 8583.981,E2 8583.981} C_VEL
LIN {X 0,Y 606.744,Z 830.79,A -85,B 0,C 180,E1 8587.978,E2 8587.978} C_VEL
LIN {X 0,Y 613.164,Z 760.379,A -85,B 0,C 180,E1 8590.501,E2 8590.501} C_VEL
LIN {X 0,Y 613.589,Z 727.811,A -85,B 0,C 180,E1 8591.326,E2 8591.326} C_VEL
LIN {X 0,Y 577.858,Z 663.19,A -85,B 0,C 180,E1 8595.867,E2 8595.867} C_VEL
LIN {X 0,Y 577.882,Z 663.19,A -85,B 0,C 180,E1 8605.75,E2 8605.75} C_VEL
LIN {X 0,Y 577.903,Z 663.19,A -85,B 0,C 180,E1 8614.862,E2 8614.862} C_VEL
LIN {X 0,Y 578.075,Z 663.19,A -85,B 0,C 180,E1 8623.231,E2 8623.231} C_VEL
LIN {X 0,Y 578.388,Z 663.19,A -85,B 0,C 180,E1 8630.162,E2 8630.162} C_VEL
LIN {X 0,Y 578.5,Z 663.19,A -85,B 0,C 180,E1 8637.728,E2 8637.728} C_VEL
LIN {X 0,Y 578.477,Z 663.19,A -85,B 0,C 180,E1 8645.253,E2 8645.253} C_VEL
LIN {X 0,Y 578.397,Z 663.19,A -85,B 0,C 180,E1 8652.872,E2 8652.872} C_VEL
LIN {X 0,Y 578.277,Z 663.19,A -85,B 0,C 180,E1 8661.421,E2 8661.421} C_VEL
LIN {X 0,Y 578.213,Z 663.19,A -85,B 0,C 180,E1 8670.769,E2 8670.769} C_VEL
LIN {X 0,Y 578.099,Z 663.19,A -85,B 0,C 180,E1 8680.013,E2 8680.013} C_VEL
LIN {X 0,Y 578.349,Z 665.237,A -85,B 0,C 180,E1 8681.375,E2 8681.375} C_VEL
LIN {X 0,Y 614.234,Z 729.761,A -85,B 0,C 180,E1 8685.943,E2 8685.943} C_VEL
LIN {X 0,Y 608.486,Z 804.364,A -85,B 0,C 180,E1 8688.215,E2 8688.215} C_VEL
LIN {X 0,Y 600.484,Z 872.973,A -85,B 0,C 180,E1 8691.88,E2 8691.88} C_VEL
LIN {X 0,Y 592.026,Z 934.025,A -85,B 0,C 180,E1 8696.898,E2 8696.898} C_VEL
LIN {X 0,Y 585.162,Z 986.012,A -85,B 0,C 180,E1 8703.191,E2 8703.191} C_VEL
LIN {X 0,Y 581.379,Z 1024.299,A -85,B 0,C 180,E1 8710.112,E2 8710.112} C_VEL
LIN {X 0,Y 579.665,Z 1048.383,A -85,B 0,C 180,E1 8717.152,E2 8717.152} C_VEL
LIN {X 0,Y 579.048,Z 1058.771,A -85,B 0,C 180,E1 8723.232,E2 8723.232} C_VEL
LIN {X 0,Y 579.206,Z 1059.775,A -85,B 0,C 180,E1 8729.25,E2 8729.25} C_VEL
LIN {X 0,Y 579.196,Z 1050.489,A -85,B 0,C 180,E1 8735.892,E2 8735.892} C_VEL
LIN {X 0,Y 580.254,Z 1030.042,A -85,B 0,C 180,E1 8742.451,E2 8742.451} C_VEL
LIN {X 0,Y 583.419,Z 997.447,A -85,B 0,C 180,E1 8748.959,E2 8748.959} C_VEL
LIN {X 0,Y 589.489,Z 950.227,A -85,B 0,C 180,E1 8755.314,E2 8755.314} C_VEL
LIN {X 0,Y 598.132,Z 890.18,A -85,B 0,C 180,E1 8760.81,E2 8760.81} C_VEL
LIN {X 0,Y 599.358,Z 880.945,A -85,B 0,C 180,E1 8761.473,E2 8761.473} C_VEL
LIN {X 0,Y 596.188,Z 854.116,A -85,B 0,C 180,E1 8763.686,E2 8763.686} C_VEL
LIN {X 0,Y 604.35,Z 783.474,A -85,B 0,C 180,E1 8766.971,E2 8766.971} C_VEL
LIN {X 0,Y 606.95,Z 730.841,A -85,B 0,C 180,E1 8768.538,E2 8768.538} C_VEL
LIN {X 0,Y 569.887,Z 663.19,A -85,B 0,C 180,E1 8773.206,E2 8773.206} C_VEL
LIN {X 0,Y 569.94,Z 663.19,A -85,B 0,C 180,E1 8781.71,E2 8781.71} C_VEL
LIN {X 0,Y 570.151,Z 663.19,A -85,B 0,C 180,E1 8790.515,E2 8790.515} C_VEL
LIN {X 0,Y 570.303,Z 663.19,A -85,B 0,C 180,E1 8798.961,E2 8798.961} C_VEL
LIN {X 0,Y 571.17,Z 663.19,A -85,B 0,C 180,E1 8808.521,E2 8808.521} C_VEL
LIN {X 0,Y 571.169,Z 663.19,A -85,B 0,C 180,E1 8817.732,E2 8817.732} C_VEL
LIN {X 0,Y 570.584,Z 663.19,A -85,B 0,C 180,E1 8826.892,E2 8826.892} C_VEL
LIN {X 0,Y 570.319,Z 663.19,A -85,B 0,C 180,E1 8834.662,E2 8834.662} C_VEL
LIN {X 0,Y 569.929,Z 663.19,A -85,B 0,C 180,E1 8843.374,E2 8843.374} C_VEL
LIN {X 0,Y 570.407,Z 663.19,A -85,B 0,C 180,E1 8851.276,E2 8851.276} C_VEL
LIN {X 0,Y 570.081,Z 663.19,A -85,B 0,C 180,E1 8860.736,E2 8860.736} C_VEL
LIN {X 0,Y 570.187,Z 664.833,A -85,B 0,C 180,E1 8863.685,E2 8863.685} C_VEL
LIN {X 0,Y 608.398,Z 734.951,A -85,B 0,C 180,E1 8868.421,E2 8868.421} C_VEL
LIN {X 0,Y 602.571,Z 809.319,A -85,B 0,C 180,E1 8870.607,E2 8870.607} C_VEL
LIN {X 0,Y 594.224,Z 878.427,A -85,B 0,C 180,E1 8874.207,E2 8874.207} C_VEL
LIN {X 0,Y 585.325,Z 940.59,A -85,B 0,C 180,E1 8879.198,E2 8879.198} C_VEL
LIN {X 0,Y 577.775,Z 993.089,A -85,B 0,C 180,E1 8885.459,E2 8885.459} C_VEL
LIN {X 0,Y 573.588,Z 1031.583,A -85,B 0,C 180,E1 8892.301,E2 8892.301} C_VEL
LIN {X 0,Y 571.712,Z 1058.416,A -85,B 0,C 180,E1 8900.073,E2 8900.073} C_VEL
LIN {X 0,Y 571.124,Z 1068.736,A -85,B 0,C 180,E1 8906.194,E2 8906.194} C_VEL
LIN {X 0,Y 571.16,Z 1069.805,A -85,B 0,C 180,E1 8912.283,E2 8912.283} C_VEL
LIN {X 0,Y 571.205,Z 1060.281,A -85,B 0,C 180,E1 8919.166,E2 8919.166} C_VEL
LIN {X 0,Y 572.395,Z 1039.874,A -85,B 0,C 180,E1 8925.757,E2 8925.757} C_VEL
LIN {X 0,Y 575.741,Z 1006.621,A -85,B 0,C 180,E1 8932.452,E2 8932.452} C_VEL
LIN {X 0,Y 582.535,Z 958.317,A -85,B 0,C 180,E1 8938.956,E2 8938.956} C_VEL
LIN {X 0,Y 591.407,Z 898.096,A -85,B 0,C 180,E1 8944.439,E2 8944.439} C_VEL
LIN {X 0,Y 600.314,Z 830.698,A -85,B 0,C 180,E1 8948.458,E2 8948.458} C_VEL
LIN {X 0,Y 607.103,Z 760.407,A -85,B 0,C 180,E1 8950.991,E2 8950.991} C_VEL
LIN {X 0,Y 607.448,Z 730.989,A -85,B 0,C 180,E1 8951.766,E2 8951.766} C_VEL
LIN {X 0,Y 570.962,Z 667.358,A -85,B 0,C 180,E1 8956.473,E2 8956.473} C_VEL
LIN {X 0,Y 569.757,Z 663.19,A -85,B 0,C 180,E1 8956.688,E2 8956.688} C_VEL
LIN {X 0,Y 569.802,Z 663.19,A -85,B 0,C 180,E1 8965.041,E2 8965.041} C_VEL
LIN {X 0,Y 569.899,Z 663.19,A -85,B 0,C 180,E1 8973.914,E2 8973.914} C_VEL
LIN {X 0,Y 570.112,Z 663.19,A -85,B 0,C 180,E1 8982.155,E2 8982.155} C_VEL
LIN {X 0,Y 570.403,Z 663.19,A -85,B 0,C 180,E1 8990.023,E2 8990.023} C_VEL
LIN {X 0,Y 570.505,Z 663.19,A -85,B 0,C 180,E1 8997.696,E2 8997.696} C_VEL
LIN {X 0,Y 570.483,Z 663.19,A -85,B 0,C 180,E1 9005.326,E2 9005.326} C_VEL
LIN {X 0,Y 570.249,Z 663.19,A -85,B 0,C 180,E1 9013.923,E2 9013.923} C_VEL
LIN {X 0,Y 570.25,Z 663.19,A -85,B 0,C 180,E1 9022.684,E2 9022.684} C_VEL
LIN {X 0,Y 570.218,Z 663.19,A -85,B 0,C 180,E1 9031.249,E2 9031.249} C_VEL
LIN {X 0,Y 570.247,Z 664.862,A -85,B 0,C 180,E1 9040.496,E2 9040.496} C_VEL
LIN {X 0,Y 608.144,Z 732.832,A -85,B 0,C 180,E1 9045.509,E2 9045.509} C_VEL
LIN {X 0,Y 601.769,Z 808.364,A -85,B 0,C 180,E1 9047.892,E2 9047.892} C_VEL
LIN {X 0,Y 593.175,Z 876.856,A -85,B 0,C 180,E1 9051.688,E2 9051.688} C_VEL
LIN {X 0,Y 584.467,Z 936.735,A -85,B 0,C 180,E1 9056.764,E2 9056.764} C_VEL
LIN {X 0,Y 577.298,Z 988.442,A -85,B 0,C 180,E1 9063.224,E2 9063.224} C_VEL
LIN {X 0,Y 573.382,Z 1026.238,A -85,B 0,C 180,E1 9070.311,E2 9070.311} C_VEL
LIN {X 0,Y 571.451,Z 1050.179,A -85,B 0,C 180,E1 9077.743,E2 9077.743} C_VEL
LIN {X 0,Y 570.863,Z 1059.801,A -85,B 0,C 180,E1 9084.665,E2 9084.665} C_VEL
LIN {X 0,Y 570.921,Z 1058.738,A -85,B 0,C 180,E1 9090.761,E2 9090.761} C_VEL
LIN {X 0,Y 571.24,Z 1048.492,A -85,B 0,C 180,E1 9096.86,E2 9096.86} C_VEL
LIN {X 0,Y 572.684,Z 1027.171,A -85,B 0,C 180,E1 9103.396,E2 9103.396} C_VEL
LIN {X 0,Y 576.73,Z 990.53,A -85,B 0,C 180,E1 9110.388,E2 9110.388} C_VEL
LIN {X 0,Y 583.902,Z 939.399,A -85,B 0,C 180,E1 9116.879,E2 9116.879} C_VEL
LIN {X 0,Y 593.048,Z 878.037,A -85,B 0,C 180,E1 9122.133,E2 9122.133} C_VEL
LIN {X 0,Y 596.188,Z 854.116,A -85,B 0,C 180,E1 9123.686,E2 9123.686} C_VEL
LIN {X 0,Y 593.644,Z 825.549,A -85,B 0,C 180,E1 9125.705,E2 9125.705} C_VEL
LIN {X 0,Y 600.833,Z 753.729,A -85,B 0,C 180,E1 9128.389,E2 9128.389} C_VEL
LIN {X 0,Y 600.438,Z 733.04,A -85,B 0,C 180,E1 9129.029,E2 9129.029} C_VEL
LIN {X 0,Y 561.949,Z 663.19,A -85,B 0,C 180,E1 9134.018,E2 9134.018} C_VEL
LIN {X 0,Y 561.906,Z 663.19,A -85,B 0,C 180,E1 9142.76,E2 9142.76} C_VEL
LIN {X 0,Y 562.114,Z 663.19,A -85,B 0,C 180,E1 9151.821,E2 9151.821} C_VEL
LIN {X 0,Y 562.238,Z 663.19,A -85,B 0,C 180,E1 9160.297,E2 9160.297} C_VEL
LIN {X 0,Y 563.154,Z 663.19,A -85,B 0,C 180,E1 9168.355,E2 9168.355} C_VEL
LIN {X 0,Y 563.161,Z 663.19,A -85,B 0,C 180,E1 9177.7,E2 9177.7} C_VEL
LIN {X 0,Y 562.552,Z 663.19,A -85,B 0,C 180,E1 9186.99,E2 9186.99} C_VEL
LIN {X 0,Y 562.264,Z 663.19,A -85,B 0,C 180,E1 9194.877,E2 9194.877} C_VEL
LIN {X 0,Y 561.957,Z 663.19,A -85,B 0,C 180,E1 9203.074,E2 9203.074} C_VEL
LIN {X 0,Y 562.362,Z 663.19,A -85,B 0,C 180,E1 9211.854,E2 9211.854} C_VEL
LIN {X 0,Y 561.965,Z 663.19,A -85,B 0,C 180,E1 9221.453,E2 9221.453} C_VEL
LIN {X 0,Y 562.191,Z 664.92,A -85,B 0,C 180,E1 9222.862,E2 9222.862} C_VEL
LIN {X 0,Y 602.243,Z 736.934,A -85,B 0,C 180,E1 9227.96,E2 9227.96} C_VEL
LIN {X 0,Y 596.014,Z 811.902,A -85,B 0,C 180,E1 9230.218,E2 9230.218} C_VEL
LIN {X 0,Y 587.21,Z 881.004,A -85,B 0,C 180,E1 9233.909,E2 9233.909} C_VEL
LIN {X 0,Y 577.817,Z 943.097,A -85,B 0,C 180,E1 9239.041,E2 9239.041} C_VEL
LIN {X 0,Y 569.967,Z 995.038,A -85,B 0,C 180,E1 9245.409,E2 9245.409} C_VEL
LIN {X 0,Y 565.592,Z 1034.247,A -85,B 0,C 180,E1 9252.66,E2 9252.66} C_VEL
LIN {X 0,Y 563.768,Z 1058.416,A -85,B 0,C 180,E1 9259.931,E2 9259.931} C_VEL
LIN {X 0,Y 563.142,Z 1068.736,A -85,B 0,C 180,E1 9266.14,E2 9266.14} C_VEL
LIN {X 0,Y 563.175,Z 1069.805,A -85,B 0,C 180,E1 9272.315,E2 9272.315} C_VEL
LIN {X 0,Y 563.235,Z 1060.281,A -85,B 0,C 180,E1 9279.297,E2 9279.297} C_VEL
LIN {X 0,Y 564.674,Z 1038.337,A -85,B 0,C 180,E1 9286.378,E2 9286.378} C_VEL
LIN {X 0,Y 568.834,Z 1002.286,A -85,B 0,C 180,E1 9293.487,E2 9293.487} C_VEL
LIN {X 0,Y 576.151,Z 952.848,A -85,B 0,C 180,E1 9299.952,E2 9299.952} C_VEL
LIN {X 0,Y 585.553,Z 891.108,A -85,B 0,C 180,E1 9305.393,E2 9305.393} C_VEL
LIN {X 0,Y 594.837,Z 823.097,A -85,B 0,C 180,E1 9309.292,E2 9309.292} C_VEL
LIN {X 0,Y 601.494,Z 755.237,A -85,B 0,C 180,E1 9311.622,E2 9311.622} C_VEL
LIN {X 0,Y 601.224,Z 733.945,A -85,B 0,C 180,E1 9312.234,E2 9312.234} C_VEL
LIN {X 0,Y 564.808,Z 669.508,A -85,B 0,C 180,E1 9317.119,E2 9317.119} C_VEL
LIN {X 0,Y 561.645,Z 663.19,A -85,B 0,C 180,E1 9317.613,E2 9317.613} C_VEL
LIN {X 0,Y 561.765,Z 663.19,A -85,B 0,C 180,E1 9326.347,E2 9326.347} C_VEL
LIN {X 0,Y 561.836,Z 663.19,A -85,B 0,C 180,E1 9335.227,E2 9335.227} C_VEL
LIN {X 0,Y 562.077,Z 663.19,A -85,B 0,C 180,E1 9343.511,E2 9343.511} C_VEL
LIN {X 0,Y 562.314,Z 663.19,A -85,B 0,C 180,E1 9351.446,E2 9351.446} C_VEL
LIN {X 0,Y 562.396,Z 663.19,A -85,B 0,C 180,E1 9359.21,E2 9359.21} C_VEL
LIN {X 0,Y 562.463,Z 663.19,A -85,B 0,C 180,E1 9365.403,E2 9365.403} C_VEL
LIN {X 0,Y 562.319,Z 663.19,A -85,B 0,C 180,E1 9373.246,E2 9373.246} C_VEL
LIN {X 0,Y 562.263,Z 663.19,A -85,B 0,C 180,E1 9381.493,E2 9381.493} C_VEL
LIN {X 0,Y 562.176,Z 663.19,A -85,B 0,C 180,E1 9389.946,E2 9389.946} C_VEL
LIN {X 0,Y 562.085,Z 663.19,A -85,B 0,C 180,E1 9399.529,E2 9399.529} C_VEL
LIN {X 0,Y 602.071,Z 735.837,A -85,B 0,C 180,E1 9405.059,E2 9405.059} C_VEL
LIN {X 0,Y 595.146,Z 811.308,A -85,B 0,C 180,E1 9407.529,E2 9407.529} C_VEL
LIN {X 0,Y 585.905,Z 880.698,A -85,B 0,C 180,E1 9411.493,E2 9411.493} C_VEL
LIN {X 0,Y 576.833,Z 940.487,A -85,B 0,C 180,E1 9416.741,E2 9416.741} C_VEL
LIN {X 0,Y 569.39,Z 991.244,A -85,B 0,C 180,E1 9423.315,E2 9423.315} C_VEL
LIN {X 0,Y 565.365,Z 1027.619,A -85,B 0,C 180,E1 9430.41,E2 9430.41} C_VEL
LIN {X 0,Y 563.528,Z 1050.089,A -85,B 0,C 180,E1 9437.568,E2 9437.568} C_VEL
LIN {X 0,Y 562.865,Z 1059.772,A -85,B 0,C 180,E1 9444.589,E2 9444.589} C_VEL
LIN {X 0,Y 562.928,Z 1058.784,A -85,B 0,C 180,E1 9450.771,E2 9450.771} C_VEL
LIN {X 0,Y 563.267,Z 1048.6,A -85,B 0,C 180,E1 9456.958,E2 9456.958} C_VEL
LIN {X 0,Y 565.05,Z 1025.699,A -85,B 0,C 180,E1 9463.977,E2 9463.977} C_VEL
LIN {X 0,Y 569.703,Z 987.028,A -85,B 0,C 180,E1 9471.245,E2 9471.245} C_VEL
LIN {X 0,Y 577.418,Z 935.596,A -85,B 0,C 180,E1 9477.692,E2 9477.692} C_VEL
LIN {X 0,Y 587.011,Z 873.751,A -85,B 0,C 180,E1 9482.907,E2 9482.907} C_VEL
LIN {X 0,Y 593.644,Z 825.549,A -85,B 0,C 180,E1 9485.705,E2 9485.705} C_VEL
LIN {X 0,Y 590.849,Z 795.538,A -85,B 0,C 180,E1 9487.518,E2 9487.518} C_VEL
LIN {X 0,Y 594.679,Z 736.914,A -85,B 0,C 180,E1 9489.424,E2 9489.424} C_VEL
LIN {X 0,Y 553.881,Z 663.19,A -85,B 0,C 180,E1 9495.06,E2 9495.06} C_VEL
LIN {X 0,Y 553.873,Z 663.19,A -85,B 0,C 180,E1 9503.923,E2 9503.923} C_VEL
LIN {X 0,Y 554.076,Z 663.19,A -85,B 0,C 180,E1 9513.148,E2 9513.148} C_VEL
LIN {X 0,Y 554.244,Z 663.19,A -85,B 0,C 180,E1 9521.662,E2 9521.662} C_VEL
LIN {X 0,Y 554.943,Z 663.19,A -85,B 0,C 180,E1 9529.777,E2 9529.777} C_VEL
LIN {X 0,Y 554.597,Z 663.19,A -85,B 0,C 180,E1 9539.233,E2 9539.233} C_VEL
LIN {X 0,Y 554.545,Z 663.19,A -85,B 0,C 180,E1 9547.092,E2 9547.092} C_VEL
LIN {X 0,Y 554.231,Z 663.19,A -85,B 0,C 180,E1 9555.097,E2 9555.097} C_VEL
LIN {X 0,Y 553.904,Z 663.19,A -85,B 0,C 180,E1 9563.492,E2 9563.492} C_VEL
LIN {X 0,Y 554.322,Z 663.19,A -85,B 0,C 180,E1 9572.291,E2 9572.291} C_VEL
LIN {X 0,Y 554.063,Z 664.305,A -85,B 0,C 180,E1 9581.975,E2 9581.975} C_VEL
LIN {X 0,Y 596.052,Z 740.067,A -85,B 0,C 180,E1 9587.513,E2 9587.513} C_VEL
LIN {X 0,Y 589.317,Z 815.338,A -85,B 0,C 180,E1 9589.855,E2 9589.855} C_VEL
LIN {X 0,Y 579.971,Z 884.76,A -85,B 0,C 180,E1 9593.694,E2 9593.694} C_VEL
LIN {X 0,Y 570.087,Z 946.521,A -85,B 0,C 180,E1 9598.979,E2 9598.979} C_VEL
LIN {X 0,Y 562.066,Z 997.846,A -85,B 0,C 180,E1 9605.493,E2 9605.493} C_VEL
LIN {X 0,Y 557.598,Z 1035.948,A -85,B 0,C 180,E1 9612.803,E2 9612.803} C_VEL
LIN {X 0,Y 555.533,Z 1060.283,A -85,B 0,C 180,E1 9620.574,E2 9620.574} C_VEL
LIN {X 0,Y 554.824,Z 1069.805,A -85,B 0,C 180,E1 9627.651,E2 9627.651} C_VEL
LIN {X 0,Y 554.992,Z 1068.736,A -85,B 0,C 180,E1 9633.917,E2 9633.917} C_VEL
LIN {X 0,Y 555.779,Z 1055.519,A -85,B 0,C 180,E1 9641.409,E2 9641.409} C_VEL
LIN {X 0,Y 558.44,Z 1027.971,A -85,B 0,C 180,E1 9649.018,E2 9649.018} C_VEL
LIN {X 0,Y 563.896,Z 986.406,A -85,B 0,C 180,E1 9656.187,E2 9656.187} C_VEL
LIN {X 0,Y 572.498,Z 931.64,A -85,B 0,C 180,E1 9662.499,E2 9662.499} C_VEL
LIN {X 0,Y 582.273,Z 868.447,A -85,B 0,C 180,E1 9667.388,E2 9667.388} C_VEL
LIN {X 0,Y 591.533,Z 796.39,A -85,B 0,C 180,E1 9670.907,E2 9670.907} C_VEL
LIN {X 0,Y 595.358,Z 737.498,A -85,B 0,C 180,E1 9672.67,E2 9672.67} C_VEL
LIN {X 0,Y 560.657,Z 675.618,A -85,B 0,C 180,E1 9677.48,E2 9677.48} C_VEL
LIN {X 0,Y 553.566,Z 663.19,A -85,B 0,C 180,E1 9678.65,E2 9678.65} C_VEL
LIN {X 0,Y 553.776,Z 663.19,A -85,B 0,C 180,E1 9687.673,E2 9687.673} C_VEL
LIN {X 0,Y 553.893,Z 663.19,A -85,B 0,C 180,E1 9696.57,E2 9696.57} C_VEL
LIN {X 0,Y 554.405,Z 663.19,A -85,B 0,C 180,E1 9706.169,E2 9706.169} C_VEL
LIN {X 0,Y 554.982,Z 663.19,A -85,B 0,C 180,E1 9716.063,E2 9716.063} C_VEL
LIN {X 0,Y 554.889,Z 663.19,A -85,B 0,C 180,E1 9724.063,E2 9724.063} C_VEL
LIN {X 0,Y 554.282,Z 663.19,A -85,B 0,C 180,E1 9733.442,E2 9733.442} C_VEL
LIN {X 0,Y 554.253,Z 663.19,A -85,B 0,C 180,E1 9741.678,E2 9741.678} C_VEL
LIN {X 0,Y 554.147,Z 663.19,A -85,B 0,C 180,E1 9750.458,E2 9750.458} C_VEL
LIN {X 0,Y 554.269,Z 665.103,A -85,B 0,C 180,E1 9758.655,E2 9758.655} C_VEL
LIN {X 0,Y 594.014,Z 734.355,A -85,B 0,C 180,E1 9764.298,E2 9764.298} C_VEL
LIN {X 0,Y 595.487,Z 748.535,A -85,B 0,C 180,E1 9764.865,E2 9764.865} C_VEL
LIN {X 0,Y 587.672,Z 821.398,A -85,B 0,C 180,E1 9767.484,E2 9767.484} C_VEL
LIN {X 0,Y 577.758,Z 890.1,A -85,B 0,C 180,E1 9771.703,E2 9771.703} C_VEL
LIN {X 0,Y 568.252,Z 948.982,A -85,B 0,C 180,E1 9777.253,E2 9777.253} C_VEL
LIN {X 0,Y 561.051,Z 996.988,A -85,B 0,C 180,E1 9783.946,E2 9783.946} C_VEL
LIN {X 0,Y 556.827,Z 1032.112,A -85,B 0,C 180,E1 9791.337,E2 9791.337} C_VEL
LIN {X 0,Y 555.293,Z 1051.58,A -85,B 0,C 180,E1 9798.181,E2 9798.181} C_VEL
LIN {X 0,Y 554.881,Z 1059.743,A -85,B 0,C 180,E1 9804.511,E2 9804.511} C_VEL
LIN {X 0,Y 554.93,Z 1058.825,A -85,B 0,C 180,E1 9810.782,E2 9810.782} C_VEL
LIN {X 0,Y 555.325,Z 1048.708,A -85,B 0,C 180,E1 9817.058,E2 9817.058} C_VEL
LIN {X 0,Y 557.197,Z 1025.895,A -85,B 0,C 180,E1 9824.178,E2 9824.178} C_VEL
LIN {X 0,Y 562.152,Z 987.238,A -85,B 0,C 180,E1 9831.563,E2 9831.563} C_VEL
LIN {X 0,Y 570.387,Z 935.328,A -85,B 0,C 180,E1 9838.153,E2 9838.153} C_VEL
LIN {X 0,Y 580.352,Z 874.063,A -85,B 0,C 180,E1 9843.366,E2 9843.366} C_VEL
LIN {X 0,Y 589.722,Z 805.795,A -85,B 0,C 180,E1 9847.104,E2 9847.104} C_VEL
LIN {X 0,Y 590.849,Z 795.538,A -85,B 0,C 180,E1 9847.518,E2 9847.518} C_VEL
LIN {X 0,Y 587.669,Z 764.351,A -85,B 0,C 180,E1 9849.118,E2 9849.118} C_VEL
LIN {X 0,Y 588.204,Z 739.348,A -85,B 0,C 180,E1 9849.915,E2 9849.915} C_VEL
LIN {X 0,Y 545.859,Z 663.19,A -85,B 0,C 180,E1 9856.059,E2 9856.059} C_VEL
LIN {X 0,Y 545.847,Z 663.19,A -85,B 0,C 180,E1 9865.269,E2 9865.269} C_VEL
LIN {X 0,Y 546.083,Z 663.19,A -85,B 0,C 180,E1 9874.5,E2 9874.5} C_VEL
LIN {X 0,Y 546.456,Z 663.19,A -85,B 0,C 180,E1 9883.209,E2 9883.209} C_VEL
LIN {X 0,Y 546.607,Z 663.19,A -85,B 0,C 180,E1 9891.233,E2 9891.233} C_VEL
LIN {X 0,Y 546.611,Z 663.19,A -85,B 0,C 180,E1 9899.222,E2 9899.222} C_VEL
LIN {X 0,Y 546.516,Z 663.19,A -85,B 0,C 180,E1 9907.197,E2 9907.197} C_VEL
LIN {X 0,Y 546.181,Z 663.19,A -85,B 0,C 180,E1 9915.325,E2 9915.325} C_VEL
LIN {X 0,Y 545.886,Z 663.19,A -85,B 0,C 180,E1 9923.795,E2 9923.795} C_VEL
LIN {X 0,Y 546.3,Z 663.19,A -85,B 0,C 180,E1 9932.825,E2 9932.825} C_VEL
LIN {X 0,Y 546.069,Z 664.396,A -85,B 0,C 180,E1 9941.076,E2 9941.076} C_VEL
LIN {X 0,Y 589.802,Z 741.995,A -85,B 0,C 180,E1 9947.02,E2 9947.02} C_VEL
LIN {X 0,Y 582.881,Z 817.023,A -85,B 0,C 180,E1 9949.422,E2 9949.422} C_VEL
LIN {X 0,Y 573.118,Z 886.102,A -85,B 0,C 180,E1 9953.31,E2 9953.31} C_VEL
LIN {X 0,Y 562.998,Z 946.437,A -85,B 0,C 180,E1 9958.543,E2 9958.543} C_VEL
LIN {X 0,Y 554.471,Z 997.764,A -85,B 0,C 180,E1 9965.135,E2 9965.135} C_VEL
LIN {X 0,Y 549.783,Z 1034.958,A -85,B 0,C 180,E1 9972.315,E2 9972.315} C_VEL
LIN {X 0,Y 547.872,Z 1058.478,A -85,B 0,C 180,E1 9979.662,E2 9979.662} C_VEL
LIN {X 0,Y 547.174,Z 1068.737,A -85,B 0,C 180,E1 9986.028,E2 9986.028} C_VEL
LIN {X 0,Y 547.166,Z 1069.805,A -85,B 0,C 180,E1 9992.383,E2 9992.383} C_VEL
LIN {X 0,Y 547.268,Z 1060.591,A -85,B 0,C 180,E1 9999.411,E2 9999.411} C_VEL
LIN {X 0,Y 548.801,Z 1039.871,A -85,B 0,C 180,E1 10006.453,E2 10006.453} C_VEL
LIN {X 0,Y 553.361,Z 1004.131,A -85,B 0,C 180,E1 10013.842,E2 10013.842} C_VEL
LIN {X 0,Y 561.611,Z 954.127,A -85,B 0,C 180,E1 10020.641,E2 10020.641} C_VEL
LIN {X 0,Y 571.923,Z 892.803,A -85,B 0,C 180,E1 10026.213,E2 10026.213} C_VEL
LIN {X 0,Y 582.148,Z 824.891,A -85,B 0,C 180,E1 10030.229,E2 10030.229} C_VEL
LIN {X 0,Y 589.665,Z 755.65,A -85,B 0,C 180,E1 10032.661,E2 10032.661} C_VEL
LIN {X 0,Y 588.956,Z 739.832,A -85,B 0,C 180,E1 10033.201,E2 10033.201} C_VEL
LIN {X 0,Y 556.224,Z 681.231,A -85,B 0,C 180,E1 10037.891,E2 10037.891} C_VEL
LIN {X 0,Y 545.566,Z 663.19,A -85,B 0,C 180,E1 10039.851,E2 10039.851} C_VEL
LIN {X 0,Y 545.819,Z 663.19,A -85,B 0,C 180,E1 10049.02,E2 10049.02} C_VEL
LIN {X 0,Y 546.054,Z 663.19,A -85,B 0,C 180,E1 10058.484,E2 10058.484} C_VEL
LIN {X 0,Y 546.52,Z 663.19,A -85,B 0,C 180,E1 10067.96,E2 10067.96} C_VEL
LIN {X 0,Y 546.997,Z 663.19,A -85,B 0,C 180,E1 10076.005,E2 10076.005} C_VEL
LIN {X 0,Y 546.95,Z 663.19,A -85,B 0,C 180,E1 10083.961,E2 10083.961} C_VEL
LIN {X 0,Y 546.265,Z 663.19,A -85,B 0,C 180,E1 10093.643,E2 10093.643} C_VEL
LIN {X 0,Y 546.218,Z 663.19,A -85,B 0,C 180,E1 10102.014,E2 10102.014} C_VEL
LIN {X 0,Y 546.12,Z 663.19,A -85,B 0,C 180,E1 10110.921,E2 10110.921} C_VEL
LIN {X 0,Y 546.15,Z 664.7,A -85,B 0,C 180,E1 10117.637,E2 10117.637} C_VEL
LIN {X 0,Y 585.627,Z 732.52,A -85,B 0,C 180,E1 10123.462,E2 10123.462} C_VEL
LIN {X 0,Y 589.735,Z 746.824,A -85,B 0,C 180,E1 10124.286,E2 10124.286} C_VEL
LIN {X 0,Y 581.671,Z 819.855,A -85,B 0,C 180,E1 10126.891,E2 10126.891} C_VEL
LIN {X 0,Y 571.528,Z 887.775,A -85,B 0,C 180,E1 10131.046,E2 10131.046} C_VEL
LIN {X 0,Y 561.495,Z 947.006,A -85,B 0,C 180,E1 10136.596,E2 10136.596} C_VEL
LIN {X 0,Y 553.58,Z 995.54,A -85,B 0,C 180,E1 10143.348,E2 10143.348} C_VEL
LIN {X 0,Y 549.023,Z 1031.934,A -85,B 0,C 180,E1 10151.062,E2 10151.062} C_VEL
LIN {X 0,Y 547.371,Z 1051.491,A -85,B 0,C 180,E1 10158.008,E2 10158.008} C_VEL
LIN {X 0,Y 546.882,Z 1059.714,A -85,B 0,C 180,E1 10164.43,E2 10164.43} C_VEL
LIN {X 0,Y 546.945,Z 1058.86,A -85,B 0,C 180,E1 10170.794,E2 10170.794} C_VEL
LIN {X 0,Y 547.657,Z 1046.9,A -85,B 0,C 180,E1 10177.958,E2 10177.958} C_VEL
LIN {X 0,Y 550.283,Z 1020.932,A -85,B 0,C 180,E1 10185.585,E2 10185.585} C_VEL
LIN {X 0,Y 556.097,Z 979.705,A -85,B 0,C 180,E1 10193.078,E2 10193.078} C_VEL
LIN {X 0,Y 564.849,Z 927.158,A -85,B 0,C 180,E1 10199.422,E2 10199.422} C_VEL
LIN {X 0,Y 575.206,Z 864.032,A -85,B 0,C 180,E1 10204.527,E2 10204.527} C_VEL
LIN {X 0,Y 584.822,Z 794.036,A -85,B 0,C 180,E1 10208.093,E2 10208.093} C_VEL
LIN {X 0,Y 587.669,Z 764.351,A -85,B 0,C 180,E1 10209.118,E2 10209.118} C_VEL
LIN {X 0,Y 583.703,Z 745.157,A -85,B 0,C 180,E1 10210.147,E2 10210.147} C_VEL
LIN {X 0,Y 578.473,Z 734.984,A -85,B 0,C 180,E1 10210.922,E2 10210.922} C_VEL
LIN {X 0,Y 537.854,Z 663.19,A -85,B 0,C 180,E1 10216.849,E2 10216.849} C_VEL
LIN {X 0,Y 537.863,Z 663.19,A -85,B 0,C 180,E1 10226.636,E2 10226.636} C_VEL
LIN {X 0,Y 538.196,Z 663.19,A -85,B 0,C 180,E1 10236.307,E2 10236.307} C_VEL
LIN {X 0,Y 538.941,Z 663.19,A -85,B 0,C 180,E1 10246.168,E2 10246.168} C_VEL
LIN {X 0,Y 538.938,Z 663.19,A -85,B 0,C 180,E1 10255.98,E2 10255.98} C_VEL
LIN {X 0,Y 538.872,Z 663.19,A -85,B 0,C 180,E1 10265.675,E2 10265.675} C_VEL
LIN {X 0,Y 538.16,Z 663.19,A -85,B 0,C 180,E1 10275.559,E2 10275.559} C_VEL
LIN {X 0,Y 537.86,Z 663.19,A -85,B 0,C 180,E1 10284.172,E2 10284.172} C_VEL
LIN {X 0,Y 538.184,Z 663.19,A -85,B 0,C 180,E1 10293.778,E2 10293.778} C_VEL
LIN {X 0,Y 538.223,Z 665.186,A -85,B 0,C 180,E1 10300.167,E2 10300.167} C_VEL
LIN {X 0,Y 582.789,Z 743.016,A -85,B 0,C 180,E1 10306.423,E2 10306.423} C_VEL
LIN {X 0,Y 576.473,Z 818.275,A -85,B 0,C 180,E1 10308.966,E2 10308.966} C_VEL
LIN {X 0,Y 566.197,Z 887.775,A -85,B 0,C 180,E1 10312.944,E2 10312.944} C_VEL
LIN {X 0,Y 555.584,Z 948.283,A -85,B 0,C 180,E1 10318.305,E2 10318.305} C_VEL
LIN {X 0,Y 546.716,Z 999.017,A -85,B 0,C 180,E1 10324.977,E2 10324.977} C_VEL
LIN {X 0,Y 541.808,Z 1036.742,A -85,B 0,C 180,E1 10332.479,E2 10332.479} C_VEL
LIN {X 0,Y 539.624,Z 1060.509,A -85,B 0,C 180,E1 10340.411,E2 10340.411} C_VEL
LIN {X 0,Y 538.863,Z 1069.805,A -85,B 0,C 180,E1 10347.581,E2 10347.581} C_VEL
LIN {X 0,Y 539.033,Z 1068.737,A -85,B 0,C 180,E1 10354.033,E2 10354.033} C_VEL
LIN {X 0,Y 539.974,Z 1055.519,A -85,B 0,C 180,E1 10361.748,E2 10361.748} C_VEL
LIN {X 0,Y 542.785,Z 1027.943,A -85,B 0,C 180,E1 10369.588,E2 10369.588} C_VEL
LIN {X 0,Y 548.902,Z 986.546,A -85,B 0,C 180,E1 10376.912,E2 10376.912} C_VEL
LIN {X 0,Y 558.497,Z 932.044,A -85,B 0,C 180,E1 10383.355,E2 10383.355} C_VEL
LIN {X 0,Y 569.259,Z 869.06,A -85,B 0,C 180,E1 10388.351,E2 10388.351} C_VEL
LIN {X 0,Y 579.27,Z 798.83,A -85,B 0,C 180,E1 10391.878,E2 10391.878} C_VEL
LIN {X 0,Y 583.279,Z 743.691,A -85,B 0,C 180,E1 10393.64,E2 10393.64} C_VEL
LIN {X 0,Y 551.985,Z 686.903,A -85,B 0,C 180,E1 10398.289,E2 10398.289} C_VEL
LIN {X 0,Y 537.592,Z 663.19,A -85,B 0,C 180,E1 10400.87,E2 10400.87} C_VEL
LIN {X 0,Y 537.847,Z 663.19,A -85,B 0,C 180,E1 10410.386,E2 10410.386} C_VEL
LIN {X 0,Y 538.06,Z 663.19,A -85,B 0,C 180,E1 10419.334,E2 10419.334} C_VEL
LIN {X 0,Y 538.488,Z 663.19,A -85,B 0,C 180,E1 10427.778,E2 10427.778} C_VEL
LIN {X 0,Y 538.994,Z 663.19,A -85,B 0,C 180,E1 10435.946,E2 10435.946} C_VEL
LIN {X 0,Y 538.937,Z 663.19,A -85,B 0,C 180,E1 10444.02,E2 10444.02} C_VEL
LIN {X 0,Y 538.233,Z 663.19,A -85,B 0,C 180,E1 10453.851,E2 10453.851} C_VEL
LIN {X 0,Y 538.172,Z 663.19,A -85,B 0,C 180,E1 10462.36,E2 10462.36} C_VEL
LIN {X 0,Y 538.095,Z 663.19,A -85,B 0,C 180,E1 10471.434,E2 10471.434} C_VEL
LIN {X 0,Y 538.234,Z 665.027,A -85,B 0,C 180,E1 10476.606,E2 10476.606} C_VEL
LIN {X 0,Y 576.746,Z 729.732,A -85,B 0,C 180,E1 10482.51,E2 10482.51} C_VEL
LIN {X 0,Y 583.827,Z 748.353,A -85,B 0,C 180,E1 10483.78,E2 10483.78} C_VEL
LIN {X 0,Y 575.377,Z 821.213,A -85,B 0,C 180,E1 10486.422,E2 10486.422} C_VEL
LIN {X 0,Y 564.948,Z 887.818,A -85,B 0,C 180,E1 10490.552,E2 10490.552} C_VEL
LIN {X 0,Y 554.301,Z 947.279,A -85,B 0,C 180,E1 10496.185,E2 10496.185} C_VEL
LIN {X 0,Y 546.035,Z 995.336,A -85,B 0,C 180,E1 10502.95,E2 10502.95} C_VEL
LIN {X 0,Y 541.181,Z 1031.978,A -85,B 0,C 180,E1 10510.838,E2 10510.838} C_VEL
LIN {X 0,Y 539.222,Z 1052.982,A -85,B 0,C 180,E1 10518.646,E2 10518.646} C_VEL
LIN {X 0,Y 538.949,Z 1060.297,A -85,B 0,C 180,E1 10525.966,E2 10525.966} C_VEL
LIN {X 0,Y 539.644,Z 1055.815,A -85,B 0,C 180,E1 10533.48,E2 10533.48} C_VEL
LIN {X 0,Y 540.39,Z 1039.064,A -85,B 0,C 180,E1 10540.967,E2 10540.967} C_VEL
LIN {X 0,Y 543.817,Z 1007.703,A -85,B 0,C 180,E1 10548.703,E2 10548.703} C_VEL
LIN {X 0,Y 551.172,Z 962.626,A -85,B 0,C 180,E1 10555.86,E2 10555.86} C_VEL
LIN {X 0,Y 561.72,Z 905.856,A -85,B 0,C 180,E1 10561.877,E2 10561.877} C_VEL
LIN {X 0,Y 572.576,Z 840.541,A -85,B 0,C 180,E1 10566.435,E2 10566.435} C_VEL
LIN {X 0,Y 581.165,Z 769.141,A -85,B 0,C 180,E1 10569.505,E2 10569.505} C_VEL
LIN {X 0,Y 582.104,Z 742.745,A -85,B 0,C 180,E1 10570.353,E2 10570.353} C_VEL
LIN {X 0,Y 578.473,Z 734.984,A -85,B 0,C 180,E1 10570.922,E2 10570.922} C_VEL
LIN {X 0,Y 564.839,Z 723.6,A -85,B 0,C 180,E1 10572.54,E2 10572.54} C_VEL
LIN {X 0,Y 529.791,Z 663.19,A -85,B 0,C 180,E1 10577.923,E2 10577.923} C_VEL
LIN {X 0,Y 529.898,Z 663.19,A -85,B 0,C 180,E1 10588.023,E2 10588.023} C_VEL
LIN {X 0,Y 530.164,Z 663.19,A -85,B 0,C 180,E1 10597.283,E2 10597.283} C_VEL
LIN {X 0,Y 531.035,Z 663.19,A -85,B 0,C 180,E1 10607.64,E2 10607.64} C_VEL
LIN {X 0,Y 531.147,Z 663.19,A -85,B 0,C 180,E1 10617.561,E2 10617.561} C_VEL
LIN {X 0,Y 530.836,Z 663.19,A -85,B 0,C 180,E1 10625.761,E2 10625.761} C_VEL
LIN {X 0,Y 530.111,Z 663.19,A -85,B 0,C 180,E1 10635.802,E2 10635.802} C_VEL
LIN {X 0,Y 529.835,Z 663.19,A -85,B 0,C 180,E1 10645.639,E2 10645.639} C_VEL
LIN {X 0,Y 530.172,Z 663.19,A -85,B 0,C 180,E1 10653.956,E2 10653.956} C_VEL
LIN {X 0,Y 530.173,Z 664.868,A -85,B 0,C 180,E1 10659.166,E2 10659.166} C_VEL
LIN {X 0,Y 573.702,Z 740.11,A -85,B 0,C 180,E1 10665.509,E2 10665.509} C_VEL
LIN {X 0,Y 577.237,Z 752.27,A -85,B 0,C 180,E1 10666.201,E2 10666.201} C_VEL
LIN {X 0,Y 568.896,Z 828.128,A -85,B 0,C 180,E1 10668.899,E2 10668.899} C_VEL
LIN {X 0,Y 558.027,Z 896.377,A -85,B 0,C 180,E1 10673.076,E2 10673.076} C_VEL
LIN {X 0,Y 547.084,Z 955.968,A -85,B 0,C 180,E1 10678.713,E2 10678.713} C_VEL
LIN {X 0,Y 538.401,Z 1005.193,A -85,B 0,C 180,E1 10685.675,E2 10685.675} C_VEL
LIN {X 0,Y 533.346,Z 1041.383,A -85,B 0,C 180,E1 10693.482,E2 10693.482} C_VEL
LIN {X 0,Y 531.382,Z 1061.849,A -85,B 0,C 180,E1 10700.97,E2 10700.97} C_VEL
LIN {X 0,Y 530.866,Z 1069.804,A -85,B 0,C 180,E1 10707.545,E2 10707.545} C_VEL
LIN {X 0,Y 531.039,Z 1068.737,A -85,B 0,C 180,E1 10714.094,E2 10714.094} C_VEL
LIN {X 0,Y 532.039,Z 1055.519,A -85,B 0,C 180,E1 10721.926,E2 10721.926} C_VEL
LIN {X 0,Y 535.011,Z 1026.931,A -85,B 0,C 180,E1 10730.089,E2 10730.089} C_VEL
LIN {X 0,Y 541.829,Z 984.018,A -85,B 0,C 180,E1 10737.669,E2 10737.669} C_VEL
LIN {X 0,Y 552.199,Z 928.828,A -85,B 0,C 180,E1 10744.142,E2 10744.142} C_VEL
LIN {X 0,Y 563.542,Z 865.691,A -85,B 0,C 180,E1 10749.087,E2 10749.087} C_VEL
LIN {X 0,Y 573.752,Z 794.478,A -85,B 0,C 180,E1 10752.589,E2 10752.589} C_VEL
LIN {X 0,Y 577.415,Z 747.03,A -85,B 0,C 180,E1 10754.113,E2 10754.113} C_VEL
LIN {X 0,Y 547.502,Z 692.2,A -85,B 0,C 180,E1 10758.733,E2 10758.733} C_VEL
LIN {X 0,Y 529.581,Z 663.19,A -85,B 0,C 180,E1 10761.948,E2 10761.948} C_VEL
LIN {X 0,Y 529.826,Z 663.19,A -85,B 0,C 180,E1 10771.772,E2 10771.772} C_VEL
LIN {X 0,Y 530.056,Z 663.19,A -85,B 0,C 180,E1 10780.755,E2 10780.755} C_VEL
LIN {X 0,Y 530.432,Z 663.19,A -85,B 0,C 180,E1 10789.263,E2 10789.263} C_VEL
LIN {X 0,Y 530.568,Z 663.19,A -85,B 0,C 180,E1 10797.523,E2 10797.523} C_VEL
LIN {X 0,Y 530.424,Z 663.19,A -85,B 0,C 180,E1 10805.73,E2 10805.73} C_VEL
LIN {X 0,Y 530.205,Z 663.19,A -85,B 0,C 180,E1 10814.065,E2 10814.065} C_VEL
LIN {X 0,Y 530.147,Z 663.19,A -85,B 0,C 180,E1 10822.718,E2 10822.718} C_VEL
LIN {X 0,Y 530.008,Z 663.19,A -85,B 0,C 180,E1 10832.431,E2 10832.431} C_VEL
LIN {X 0,Y 530.322,Z 665.243,A -85,B 0,C 180,E1 10835.516,E2 10835.516} C_VEL
LIN {X 0,Y 567.905,Z 727.122,A -85,B 0,C 180,E1 10841.518,E2 10841.518} C_VEL
LIN {X 0,Y 577.796,Z 752.194,A -85,B 0,C 180,E1 10843.323,E2 10843.323} C_VEL
LIN {X 0,Y 568.726,Z 825.729,A -85,B 0,C 180,E1 10846.1,E2 10846.1} C_VEL
LIN {X 0,Y 557.458,Z 892.492,A -85,B 0,C 180,E1 10850.405,E2 10850.405} C_VEL
LIN {X 0,Y 546.329,Z 951.682,A -85,B 0,C 180,E1 10856.259,E2 10856.259} C_VEL
LIN {X 0,Y 537.848,Z 999.499,A -85,B 0,C 180,E1 10863.315,E2 10863.315} C_VEL
LIN {X 0,Y 533.133,Z 1033.149,A -85,B 0,C 180,E1 10870.907,E2 10870.907} C_VEL
LIN {X 0,Y 531.284,Z 1052.893,A -85,B 0,C 180,E1 10878.475,E2 10878.475} C_VEL
LIN {X 0,Y 530.939,Z 1060.287,A -85,B 0,C 180,E1 10885.905,E2 10885.905} C_VEL
LIN {X 0,Y 531.645,Z 1055.883,A -85,B 0,C 180,E1 10893.532,E2 10893.532} C_VEL
LIN {X 0,Y 532.426,Z 1038.05,A -85,B 0,C 180,E1 10901.5,E2 10901.5} C_VEL
LIN {X 0,Y 536.215,Z 1006.965,A -85,B 0,C 180,E1 10909.193,E2 10909.193} C_VEL
LIN {X 0,Y 543.986,Z 962.291,A -85,B 0,C 180,E1 10916.337,E2 10916.337} C_VEL
LIN {X 0,Y 555.071,Z 905.266,A -85,B 0,C 180,E1 10922.421,E2 10922.421} C_VEL
LIN {X 0,Y 566.224,Z 840.733,A -85,B 0,C 180,E1 10926.945,E2 10926.945} C_VEL
LIN {X 0,Y 575.269,Z 768.688,A -85,B 0,C 180,E1 10930.05,E2 10930.05} C_VEL
LIN {X 0,Y 575.993,Z 745.91,A -85,B 0,C 180,E1 10930.81,E2 10930.81} C_VEL
LIN {X 0,Y 564.839,Z 723.6,A -85,B 0,C 180,E1 10932.54,E2 10932.54} C_VEL
LIN {X 0,Y 546.358,Z 704.095,A -85,B 0,C 180,E1 10934.947,E2 10934.947} C_VEL
LIN {X 0,Y 521.732,Z 663.19,A -85,B 0,C 180,E1 10938.867,E2 10938.867} C_VEL
LIN {X 0,Y 521.876,Z 663.19,A -85,B 0,C 180,E1 10949.001,E2 10949.001} C_VEL
LIN {X 0,Y 522.144,Z 663.19,A -85,B 0,C 180,E1 10958.713,E2 10958.713} C_VEL
LIN {X 0,Y 522.997,Z 663.19,A -85,B 0,C 180,E1 10967.447,E2 10967.447} C_VEL
LIN {X 0,Y 523.145,Z 663.19,A -85,B 0,C 180,E1 10977.524,E2 10977.524} C_VEL
LIN {X 0,Y 522.814,Z 663.19,A -85,B 0,C 180,E1 10985.85,E2 10985.85} C_VEL
LIN {X 0,Y 522.292,Z 663.19,A -85,B 0,C 180,E1 10994.319,E2 10994.319} C_VEL
LIN {X 0,Y 521.791,Z 663.19,A -85,B 0,C 180,E1 11003.732,E2 11003.732} C_VEL
LIN {X 0,Y 522.163,Z 663.19,A -85,B 0,C 180,E1 11012.552,E2 11012.552} C_VEL
LIN {X 0,Y 522.182,Z 665.002,A -85,B 0,C 180,E1 11018.13,E2 11018.13} C_VEL
LIN {X 0,Y 564.299,Z 736.553,A -85,B 0,C 180,E1 11024.504,E2 11024.504} C_VEL
LIN {X 0,Y 571.193,Z 754.245,A -85,B 0,C 180,E1 11025.705,E2 11025.705} C_VEL
LIN {X 0,Y 562.525,Z 829.397,A -85,B 0,C 180,E1 11028.428,E2 11028.428} C_VEL
LIN {X 0,Y 551.318,Z 896.828,A -85,B 0,C 180,E1 11032.61,E2 11032.61} C_VEL
LIN {X 0,Y 539.912,Z 956.207,A -85,B 0,C 180,E1 11038.294,E2 11038.294} C_VEL
LIN {X 0,Y 530.716,Z 1005.321,A -85,B 0,C 180,E1 11045.339,E2 11045.339} C_VEL
LIN {X 0,Y 525.519,Z 1041.303,A -85,B 0,C 180,E1 11053.229,E2 11053.229} C_VEL
LIN {X 0,Y 523.442,Z 1061.849,A -85,B 0,C 180,E1 11060.832,E2 11060.832} C_VEL
LIN {X 0,Y 522.872,Z 1069.804,A -85,B 0,C 180,E1 11067.507,E2 11067.507} C_VEL
LIN {X 0,Y 523.051,Z 1068.737,A -85,B 0,C 180,E1 11074.157,E2 11074.157} C_VEL
LIN {X 0,Y 524.127,Z 1055.506,A -85,B 0,C 180,E1 11082.109,E2 11082.109} C_VEL
LIN {X 0,Y 527.16,Z 1027.251,A -85,B 0,C 180,E1 11090.311,E2 11090.311} C_VEL
LIN {X 0,Y 534.247,Z 985.008,A -85,B 0,C 180,E1 11097.927,E2 11097.927} C_VEL
LIN {X 0,Y 545.155,Z 929.882,A -85,B 0,C 180,E1 11104.525,E2 11104.525} C_VEL
LIN {X 0,Y 557.13,Z 866.396,A -85,B 0,C 180,E1 11109.581,E2 11109.581} C_VEL
LIN {X 0,Y 567.833,Z 794.805,A -85,B 0,C 180,E1 11113.14,E2 11113.14} C_VEL
LIN {X 0,Y 571.411,Z 750.218,A -85,B 0,C 180,E1 11114.609,E2 11114.609} C_VEL
LIN {X 0,Y 543.064,Z 697.395,A -85,B 0,C 180,E1 11119.186,E2 11119.186} C_VEL
LIN {X 0,Y 521.514,Z 663.19,A -85,B 0,C 180,E1 11123.095,E2 11123.095} C_VEL
LIN {X 0,Y 521.758,Z 663.19,A -85,B 0,C 180,E1 11132.43,E2 11132.43} C_VEL
LIN {X 0,Y 521.988,Z 663.19,A -85,B 0,C 180,E1 11142.204,E2 11142.204} C_VEL
LIN {X 0,Y 522.34,Z 663.19,A -85,B 0,C 180,E1 11150.786,E2 11150.786} C_VEL
LIN {X 0,Y 522.444,Z 663.19,A -85,B 0,C 180,E1 11159.15,E2 11159.15} C_VEL
LIN {X 0,Y 522.428,Z 663.19,A -85,B 0,C 180,E1 11165.818,E2 11165.818} C_VEL
LIN {X 0,Y 522.193,Z 663.19,A -85,B 0,C 180,E1 11174.285,E2 11174.285} C_VEL
LIN {X 0,Y 522.097,Z 663.19,A -85,B 0,C 180,E1 11183.088,E2 11183.088} C_VEL
LIN {X 0,Y 522.003,Z 663.19,A -85,B 0,C 180,E1 11192.52,E2 11192.52} C_VEL
LIN {X 0,Y 522.243,Z 664.999,A -85,B 0,C 180,E1 11194.328,E2 11194.328} C_VEL
LIN {X 0,Y 559.714,Z 725.703,A -85,B 0,C 180,E1 11200.581,E2 11200.581} C_VEL
LIN {X 0,Y 571.905,Z 754.674,A -85,B 0,C 180,E1 11202.819,E2 11202.819} C_VEL
LIN {X 0,Y 562.428,Z 827.356,A -85,B 0,C 180,E1 11205.63,E2 11205.63} C_VEL
LIN {X 0,Y 550.589,Z 894.198,A -85,B 0,C 180,E1 11210.02,E2 11210.02} C_VEL
LIN {X 0,Y 538.916,Z 953.289,A -85,B 0,C 180,E1 11215.995,E2 11215.995} C_VEL
LIN {X 0,Y 530.23,Z 999.634,A -85,B 0,C 180,E1 11222.965,E2 11222.965} C_VEL
LIN {X 0,Y 525.057,Z 1034.515,A -85,B 0,C 180,E1 11231.039,E2 11231.039} C_VEL
LIN {X 0,Y 523.173,Z 1054.248,A -85,B 0,C 180,E1 11239.14,E2 11239.14} C_VEL
LIN {X 0,Y 522.945,Z 1060.278,A -85,B 0,C 180,E1 11245.842,E2 11245.842} C_VEL
LIN {X 0,Y 523.57,Z 1056.338,A -85,B 0,C 180,E1 11253.32,E2 11253.32} C_VEL
LIN {X 0,Y 524.465,Z 1038.268,A -85,B 0,C 180,E1 11261.677,E2 11261.677} C_VEL
LIN {X 0,Y 528.501,Z 1007.29,A -85,B 0,C 180,E1 11269.484,E2 11269.484} C_VEL
LIN {X 0,Y 536.555,Z 963.437,A -85,B 0,C 180,E1 11276.629,E2 11276.629} C_VEL
LIN {X 0,Y 548.027,Z 906.894,A -85,B 0,C 180,E1 11282.772,E2 11282.772} C_VEL
LIN {X 0,Y 559.687,Z 842.43,A -85,B 0,C 180,E1 11287.379,E2 11287.379} C_VEL
LIN {X 0,Y 569.143,Z 770.376,A -85,B 0,C 180,E1 11290.546,E2 11290.546} C_VEL
LIN {X 0,Y 569.775,Z 748.719,A -85,B 0,C 180,E1 11291.303,E2 11291.303} C_VEL
LIN {X 0,Y 546.358,Z 704.095,A -85,B 0,C 180,E1 11294.947,E2 11294.947} C_VEL
LIN {X 0,Y 527.568,Z 686.145,A -85,B 0,C 180,E1 11297.549,E2 11297.549} C_VEL
LIN {X 0,Y 513.619,Z 663.19,A -85,B 0,C 180,E1 11300.112,E2 11300.112} C_VEL
LIN {X 0,Y 513.874,Z 663.19,A -85,B 0,C 180,E1 11308.898,E2 11308.898} C_VEL
LIN {X 0,Y 514.106,Z 663.19,A -85,B 0,C 180,E1 11318.364,E2 11318.364} C_VEL
LIN {X 0,Y 514.969,Z 663.19,A -85,B 0,C 180,E1 11327.248,E2 11327.248} C_VEL
LIN {X 0,Y 515.131,Z 663.19,A -85,B 0,C 180,E1 11337.485,E2 11337.485} C_VEL
LIN {X 0,Y 514.779,Z 663.19,A -85,B 0,C 180,E1 11345.942,E2 11345.942} C_VEL
LIN {X 0,Y 514.234,Z 663.19,A -85,B 0,C 180,E1 11354.549,E2 11354.549} C_VEL
LIN {X 0,Y 513.804,Z 663.19,A -85,B 0,C 180,E1 11363.523,E2 11363.523} C_VEL
LIN {X 0,Y 514.133,Z 663.19,A -85,B 0,C 180,E1 11373.125,E2 11373.125} C_VEL
LIN {X 0,Y 514.123,Z 664.685,A -85,B 0,C 180,E1 11377.019,E2 11377.019} C_VEL
LIN {X 0,Y 554.6,Z 732.644,A -85,B 0,C 180,E1 11383.407,E2 11383.407} C_VEL
LIN {X 0,Y 565.061,Z 757.835,A -85,B 0,C 180,E1 11385.24,E2 11385.24} C_VEL
LIN {X 0,Y 555.832,Z 833.004,A -85,B 0,C 180,E1 11388.056,E2 11388.056} C_VEL
LIN {X 0,Y 543.902,Z 900.801,A -85,B 0,C 180,E1 11392.419,E2 11392.419} C_VEL
LIN {X 0,Y 532.222,Z 959.083,A -85,B 0,C 180,E1 11398.19,E2 11398.19} C_VEL
LIN {X 0,Y 522.984,Z 1006.239,A -85,B 0,C 180,E1 11405.138,E2 11405.138} C_VEL
LIN {X 0,Y 517.615,Z 1041.562,A -85,B 0,C 180,E1 11413.061,E2 11413.061} C_VEL
LIN {X 0,Y 515.488,Z 1061.799,A -85,B 0,C 180,E1 11420.689,E2 11420.689} C_VEL
LIN {X 0,Y 514.875,Z 1069.804,A -85,B 0,C 180,E1 11427.468,E2 11427.468} C_VEL
LIN {X 0,Y 515.058,Z 1068.736,A -85,B 0,C 180,E1 11434.221,E2 11434.221} C_VEL
LIN {X 0,Y 516.2,Z 1055.426,A -85,B 0,C 180,E1 11442.297,E2 11442.297} C_VEL
LIN {X 0,Y 519.327,Z 1027.584,A -85,B 0,C 180,E1 11450.536,E2 11450.536} C_VEL
LIN {X 0,Y 526.888,Z 984.924,A -85,B 0,C 180,E1 11458.352,E2 11458.352} C_VEL
LIN {X 0,Y 538.261,Z 930.185,A -85,B 0,C 180,E1 11464.999,E2 11464.999} C_VEL
LIN {X 0,Y 550.58,Z 867.986,A -85,B 0,C 180,E1 11470.025,E2 11470.025} C_VEL
LIN {X 0,Y 561.785,Z 797.133,A -85,B 0,C 180,E1 11473.626,E2 11473.626} C_VEL
LIN {X 0,Y 565.477,Z 753.38,A -85,B 0,C 180,E1 11475.114,E2 11475.114} C_VEL
LIN {X 0,Y 537.376,Z 700.344,A -85,B 0,C 180,E1 11479.862,E2 11479.862} C_VEL
LIN {X 0,Y 513.495,Z 663.19,A -85,B 0,C 180,E1 11484.303,E2 11484.303} C_VEL
LIN {X 0,Y 513.77,Z 663.19,A -85,B 0,C 180,E1 11492.727,E2 11492.727} C_VEL
LIN {X 0,Y 513.976,Z 663.19,A -85,B 0,C 180,E1 11501.917,E2 11501.917} C_VEL
LIN {X 0,Y 514.347,Z 663.19,A -85,B 0,C 180,E1 11510.991,E2 11510.991} C_VEL
LIN {X 0,Y 514.444,Z 663.19,A -85,B 0,C 180,E1 11519.136,E2 11519.136} C_VEL
LIN {X 0,Y 514.41,Z 663.19,A -85,B 0,C 180,E1 11525.909,E2 11525.909} C_VEL
LIN {X 0,Y 514.167,Z 663.19,A -85,B 0,C 180,E1 11534.513,E2 11534.513} C_VEL
LIN {X 0,Y 514.069,Z 663.19,A -85,B 0,C 180,E1 11543.47,E2 11543.47} C_VEL
LIN {X 0,Y 514.202,Z 664.963,A -85,B 0,C 180,E1 11553.076,E2 11553.076} C_VEL
LIN {X 0,Y 551.14,Z 723.729,A -85,B 0,C 180,E1 11559.534,E2 11559.534} C_VEL
LIN {X 0,Y 565.886,Z 758.513,A -85,B 0,C 180,E1 11562.355,E2 11562.355} C_VEL
LIN {X 0,Y 555.851,Z 830.995,A -85,B 0,C 180,E1 11565.26,E2 11565.26} C_VEL
LIN {X 0,Y 543.28,Z 898.359,A -85,B 0,C 180,E1 11569.832,E2 11569.832} C_VEL
LIN {X 0,Y 531.168,Z 956.572,A -85,B 0,C 180,E1 11575.924,E2 11575.924} C_VEL
LIN {X 0,Y 522.121,Z 1003.119,A -85,B 0,C 180,E1 11583.245,E2 11583.245} C_VEL
LIN {X 0,Y 517.003,Z 1035.789,A -85,B 0,C 180,E1 11591.177,E2 11591.177} C_VEL
LIN {X 0,Y 515.216,Z 1054.217,A -85,B 0,C 180,E1 11598.97,E2 11598.97} C_VEL
LIN {X 0,Y 514.934,Z 1060.268,A -85,B 0,C 180,E1 11605.778,E2 11605.778} C_VEL
LIN {X 0,Y 515.572,Z 1056.423,A -85,B 0,C 180,E1 11613.372,E2 11613.372} C_VEL
LIN {X 0,Y 516.514,Z 1038.498,A -85,B 0,C 180,E1 11621.859,E2 11621.859} C_VEL
LIN {X 0,Y 520.669,Z 1008.679,A -85,B 0,C 180,E1 11629.568,E2 11629.568} C_VEL
LIN {X 0,Y 529.153,Z 964.535,A -85,B 0,C 180,E1 11636.933,E2 11636.933} C_VEL
LIN {X 0,Y 541.256,Z 907.368,A -85,B 0,C 180,E1 11643.235,E2 11643.235} C_VEL
LIN {X 0,Y 553.419,Z 842.577,A -85,B 0,C 180,E1 11647.91,E2 11647.91} C_VEL
LIN {X 0,Y 563.228,Z 770.723,A -85,B 0,C 180,E1 11651.091,E2 11651.091} C_VEL
LIN {X 0,Y 563.509,Z 751.48,A -85,B 0,C 180,E1 11651.816,E2 11651.816} C_VEL
LIN {X 0,Y 527.568,Z 686.145,A -85,B 0,C 180,E1 11657.549,E2 11657.549} C_VEL
LIN {X 0,Y 514.135,Z 677.475,A -85,B 0,C 180,E1 11659.518,E2 11659.518} C_VEL
LIN {X 0,Y 505.63,Z 663.19,A -85,B 0,C 180,E1 11661.402,E2 11661.402} C_VEL
LIN {X 0,Y 505.884,Z 663.19,A -85,B 0,C 180,E1 11670.349,E2 11670.349} C_VEL
LIN {X 0,Y 506.084,Z 663.19,A -85,B 0,C 180,E1 11679.845,E2 11679.845} C_VEL
LIN {X 0,Y 506.939,Z 663.19,A -85,B 0,C 180,E1 11688.797,E2 11688.797} C_VEL
LIN {X 0,Y 506.672,Z 663.19,A -85,B 0,C 180,E1 11699.16,E2 11699.16} C_VEL
LIN {X 0,Y 506.418,Z 663.19,A -85,B 0,C 180,E1 11707.77,E2 11707.77} C_VEL
LIN {X 0,Y 506.01,Z 663.19,A -85,B 0,C 180,E1 11716.576,E2 11716.576} C_VEL
LIN {X 0,Y 505.795,Z 663.19,A -85,B 0,C 180,E1 11725.813,E2 11725.813} C_VEL
LIN {X 0,Y 506.015,Z 663.19,A -85,B 0,C 180,E1 11735.47,E2 11735.47} C_VEL
LIN {X 0,Y 518.207,Z 683.271,A -85,B 0,C 180,E1 11737.986,E2 11737.986} C_VEL
LIN {X 0,Y 555.597,Z 749.632,A -85,B 0,C 180,E1 11744.02,E2 11744.02} C_VEL
LIN {X 0,Y 558.932,Z 761.74,A -85,B 0,C 180,E1 11744.773,E2 11744.773} C_VEL
LIN {X 0,Y 549.183,Z 835.987,A -85,B 0,C 180,E1 11747.661,E2 11747.661} C_VEL
LIN {X 0,Y 536.823,Z 903.11,A -85,B 0,C 180,E1 11752.093,E2 11752.093} C_VEL
LIN {X 0,Y 524.569,Z 961.612,A -85,B 0,C 180,E1 11758.042,E2 11758.042} C_VEL
LIN {X 0,Y 515.154,Z 1007.924,A -85,B 0,C 180,E1 11765.074,E2 11765.074} C_VEL
LIN {X 0,Y 509.526,Z 1042.975,A -85,B 0,C 180,E1 11773.215,E2 11773.215} C_VEL
LIN {X 0,Y 507.295,Z 1063.45,A -85,B 0,C 180,E1 11781.489,E2 11781.489} C_VEL
LIN {X 0,Y 507.038,Z 1070.269,A -85,B 0,C 180,E1 11789.144,E2 11789.144} C_VEL
LIN {X 0,Y 507.519,Z 1065.824,A -85,B 0,C 180,E1 11796.865,E2 11796.865} C_VEL
LIN {X 0,Y 508.509,Z 1048.185,A -85,B 0,C 180,E1 11805.126,E2 11805.126} C_VEL
LIN {X 0,Y 512.697,Z 1018.609,A -85,B 0,C 180,E1 11812.843,E2 11812.843} C_VEL
LIN {X 0,Y 521.741,Z 974.241,A -85,B 0,C 180,E1 11820.332,E2 11820.332} C_VEL
LIN {X 0,Y 534.432,Z 916.47,A -85,B 0,C 180,E1 11826.828,E2 11826.828} C_VEL
LIN {X 0,Y 547.366,Z 852.752,A -85,B 0,C 180,E1 11831.514,E2 11831.514} C_VEL
LIN {X 0,Y 558.212,Z 781.42,A -85,B 0,C 180,E1 11834.761,E2 11834.761} C_VEL
LIN {X 0,Y 559.514,Z 756.252,A -85,B 0,C 180,E1 11835.649,E2 11835.649} C_VEL
LIN {X 0,Y 532.489,Z 704.987,A -85,B 0,C 180,E1 11840.418,E2 11840.418} C_VEL
LIN {X 0,Y 505.479,Z 663.19,A -85,B 0,C 180,E1 11845.588,E2 11845.588} C_VEL
LIN {X 0,Y 505.736,Z 663.19,A -85,B 0,C 180,E1 11854.183,E2 11854.183} C_VEL
LIN {X 0,Y 506.012,Z 663.19,A -85,B 0,C 180,E1 11863.425,E2 11863.425} C_VEL
LIN {X 0,Y 506.425,Z 663.19,A -85,B 0,C 180,E1 11872.23,E2 11872.23} C_VEL
LIN {X 0,Y 506.641,Z 663.19,A -85,B 0,C 180,E1 11880.84,E2 11880.84} C_VEL
LIN {X 0,Y 506.487,Z 663.19,A -85,B 0,C 180,E1 11889.468,E2 11889.468} C_VEL
LIN {X 0,Y 506.211,Z 663.19,A -85,B 0,C 180,E1 11899.33,E2 11899.33} C_VEL
LIN {X 0,Y 505.96,Z 663.19,A -85,B 0,C 180,E1 11909.646,E2 11909.646} C_VEL
LIN {X 0,Y 506.13,Z 664.907,A -85,B 0,C 180,E1 11911.734,E2 11911.734} C_VEL
LIN {X 0,Y 542.997,Z 722.23,A -85,B 0,C 180,E1 11918.499,E2 11918.499} C_VEL
LIN {X 0,Y 560.135,Z 760.03,A -85,B 0,C 180,E1 11921.81,E2 11921.81} C_VEL
LIN {X 0,Y 549.584,Z 832.871,A -85,B 0,C 180,E1 11924.782,E2 11924.782} C_VEL
LIN {X 0,Y 536.742,Z 898.658,A -85,B 0,C 180,E1 11929.306,E2 11929.306} C_VEL
LIN {X 0,Y 524.203,Z 956.327,A -85,B 0,C 180,E1 11935.409,E2 11935.409} C_VEL
LIN {X 0,Y 514.553,Z 1002.942,A -85,B 0,C 180,E1 11942.819,E2 11942.819} C_VEL
LIN {X 0,Y 509.218,Z 1035.715,A -85,B 0,C 180,E1 11950.878,E2 11950.878} C_VEL
LIN {X 0,Y 507.243,Z 1054.228,A -85,B 0,C 180,E1 11958.795,E2 11958.795} C_VEL
LIN {X 0,Y 506.925,Z 1060.329,A -85,B 0,C 180,E1 11965.711,E2 11965.711} C_VEL
LIN {X 0,Y 507.605,Z 1056.568,A -85,B 0,C 180,E1 11973.425,E2 11973.425} C_VEL
LIN {X 0,Y 508.554,Z 1040.041,A -85,B 0,C 180,E1 11981.611,E2 11981.611} C_VEL
LIN {X 0,Y 512.787,Z 1010.348,A -85,B 0,C 180,E1 11989.597,E2 11989.597} C_VEL
LIN {X 0,Y 521.42,Z 967.257,A -85,B 0,C 180,E1 11997.018,E2 11997.018} C_VEL
LIN {X 0,Y 533.627,Z 911.694,A -85,B 0,C 180,E1 12003.356,E2 12003.356} C_VEL
LIN {X 0,Y 546.375,Z 847.204,A -85,B 0,C 180,E1 12008.184,E2 12008.184} C_VEL
LIN {X 0,Y 556.814,Z 775.5,A -85,B 0,C 180,E1 12011.503,E2 12011.503} C_VEL
LIN {X 0,Y 557.524,Z 754.903,A -85,B 0,C 180,E1 12012.293,E2 12012.293} C_VEL
LIN {X 0,Y 522.078,Z 689.616,A -85,B 0,C 180,E1 12018.184,E2 12018.184} C_VEL
LIN {X 0,Y 514.135,Z 677.475,A -85,B 0,C 180,E1 12019.518,E2 12019.518} C_VEL
LIN {X 0,Y 501.033,Z 669.741,A -85,B 0,C 180,E1 12021.613,E2 12021.613} C_VEL
LIN {X 0,Y 497.644,Z 663.19,A -85,B 0,C 180,E1 12022.371,E2 12022.371} C_VEL
LIN {X 0,Y 497.869,Z 663.19,A -85,B 0,C 180,E1 12031.823,E2 12031.823} C_VEL
LIN {X 0,Y 498.153,Z 663.19,A -85,B 0,C 180,E1 12041.362,E2 12041.362} C_VEL
LIN {X 0,Y 498.699,Z 663.19,A -85,B 0,C 180,E1 12050.383,E2 12050.383} C_VEL
LIN {X 0,Y 498.673,Z 663.19,A -85,B 0,C 180,E1 12059.147,E2 12059.147} C_VEL
LIN {X 0,Y 498.395,Z 663.19,A -85,B 0,C 180,E1 12067.896,E2 12067.896} C_VEL
LIN {X 0,Y 497.998,Z 663.19,A -85,B 0,C 180,E1 12076.85,E2 12076.85} C_VEL
LIN {X 0,Y 497.783,Z 663.19,A -85,B 0,C 180,E1 12086.26,E2 12086.26} C_VEL
LIN {X 0,Y 498.277,Z 665.208,A -85,B 0,C 180,E1 12094.669,E2 12094.669} C_VEL
LIN {X 0,Y 536.6,Z 726.895,A -85,B 0,C 180,E1 12101.254,E2 12101.254} C_VEL
LIN {X 0,Y 553.051,Z 763.114,A -85,B 0,C 180,E1 12104.23,E2 12104.23} C_VEL
LIN {X 0,Y 542.829,Z 837.41,A -85,B 0,C 180,E1 12107.175,E2 12107.175} C_VEL
LIN {X 0,Y 529.757,Z 905.406,A -85,B 0,C 180,E1 12111.757,E2 12111.757} C_VEL
LIN {X 0,Y 517.067,Z 963.529,A -85,B 0,C 180,E1 12117.816,E2 12117.816} C_VEL
LIN {X 0,Y 507.137,Z 1010.902,A -85,B 0,C 180,E1 12125.253,E2 12125.253} C_VEL
LIN {X 0,Y 501.161,Z 1045.418,A -85,B 0,C 180,E1 12133.747,E2 12133.747} C_VEL
LIN {X 0,Y 499.189,Z 1064.523,A -85,B 0,C 180,E1 12142.144,E2 12142.144} C_VEL
LIN {X 0,Y 499.034,Z 1070.191,A -85,B 0,C 180,E1 12149.13,E2 12149.13} C_VEL
LIN {X 0,Y 499.504,Z 1065.745,A -85,B 0,C 180,E1 12156.975,E2 12156.975} C_VEL
LIN {X 0,Y 500.608,Z 1048.104,A -85,B 0,C 180,E1 12165.37,E2 12165.37} C_VEL
LIN {X 0,Y 505.048,Z 1018.437,A -85,B 0,C 180,E1 12173.228,E2 12173.228} C_VEL
LIN {X 0,Y 514.535,Z 974.242,A -85,B 0,C 180,E1 12180.802,E2 12180.802} C_VEL
LIN {X 0,Y 527.933,Z 916.21,A -85,B 0,C 180,E1 12187.397,E2 12187.397} C_VEL
LIN {X 0,Y 541.497,Z 852.048,A -85,B 0,C 180,E1 12192.137,E2 12192.137} C_VEL
LIN {X 0,Y 552.694,Z 781.054,A -85,B 0,C 180,E1 12195.367,E2 12195.367} C_VEL
LIN {X 0,Y 553.757,Z 759.647,A -85,B 0,C 180,E1 12196.159,E2 12196.159} C_VEL
LIN {X 0,Y 526.678,Z 707.697,A -85,B 0,C 180,E1 12201.163,E2 12201.163} C_VEL
LIN {X 0,Y 497.518,Z 663.19,A -85,B 0,C 180,E1 12206.95,E2 12206.95} C_VEL
LIN {X 0,Y 497.681,Z 663.19,A -85,B 0,C 180,E1 12215.667,E2 12215.667} C_VEL
LIN {X 0,Y 498.137,Z 663.19,A -85,B 0,C 180,E1 12224.97,E2 12224.97} C_VEL
LIN {X 0,Y 498.948,Z 663.19,A -85,B 0,C 180,E1 12235.62,E2 12235.62} C_VEL
LIN {X 0,Y 498.802,Z 663.19,A -85,B 0,C 180,E1 12244.344,E2 12244.344} C_VEL
LIN {X 0,Y 498.247,Z 663.19,A -85,B 0,C 180,E1 12253.188,E2 12253.188} C_VEL
LIN {X 0,Y 498.045,Z 663.19,A -85,B 0,C 180,E1 12262.371,E2 12262.371} C_VEL
LIN {X 0,Y 498.134,Z 664.967,A -85,B 0,C 180,E1 12270.314,E2 12270.314} C_VEL
LIN {X 0,Y 534.02,Z 719.53,A -85,B 0,C 180,E1 12277.26,E2 12277.26} C_VEL
LIN {X 0,Y 554.211,Z 763.208,A -85,B 0,C 180,E1 12281.302,E2 12281.302} C_VEL
LIN {X 0,Y 543.26,Z 835.383,A -85,B 0,C 180,E1 12284.329,E2 12284.329} C_VEL
LIN {X 0,Y 529.783,Z 901.231,A -85,B 0,C 180,E1 12288.964,E2 12288.964} C_VEL
LIN {X 0,Y 516.559,Z 959.091,A -85,B 0,C 180,E1 12295.268,E2 12295.268} C_VEL
LIN {X 0,Y 506.631,Z 1004.973,A -85,B 0,C 180,E1 12302.841,E2 12302.841} C_VEL
LIN {X 0,Y 500.872,Z 1038.336,A -85,B 0,C 180,E1 12311.464,E2 12311.464} C_VEL
LIN {X 0,Y 499.201,Z 1055.45,A -85,B 0,C 180,E1 12319.498,E2 12319.498} C_VEL
LIN {X 0,Y 499.264,Z 1060.485,A -85,B 0,C 180,E1 12327.784,E2 12327.784} C_VEL
LIN {X 0,Y 499.459,Z 1054.325,A -85,B 0,C 180,E1 12335.226,E2 12335.226} C_VEL
LIN {X 0,Y 500.92,Z 1036.326,A -85,B 0,C 180,E1 12343.123,E2 12343.123} C_VEL
LIN {X 0,Y 506.074,Z 1005.07,A -85,B 0,C 180,E1 12351.073,E2 12351.073} C_VEL
LIN {X 0,Y 515.997,Z 959.811,A -85,B 0,C 180,E1 12358.508,E2 12358.508} C_VEL
LIN {X 0,Y 528.959,Z 902.804,A -85,B 0,C 180,E1 12364.699,E2 12364.699} C_VEL
LIN {X 0,Y 541.945,Z 837.559,A -85,B 0,C 180,E1 12369.303,E2 12369.303} C_VEL
LIN {X 0,Y 552.31,Z 764.972,A -85,B 0,C 180,E1 12372.406,E2 12372.406} C_VEL
LIN {X 0,Y 545.859,Z 746.313,A -85,B 0,C 180,E1 12373.812,E2 12373.812} C_VEL
LIN {X 0,Y 512.769,Z 687.465,A -85,B 0,C 180,E1 12379.489,E2 12379.489} C_VEL
LIN {X 0,Y 501.033,Z 669.741,A -85,B 0,C 180,E1 12381.613,E2 12381.613} C_VEL
LIN {X 0,Y 489.645,Z 663.19,A -85,B 0,C 180,E1 12383.934,E2 12383.934} C_VEL
LIN {X 0,Y 489.854,Z 663.19,A -85,B 0,C 180,E1 12393.324,E2 12393.324} C_VEL
LIN {X 0,Y 490.279,Z 663.19,A -85,B 0,C 180,E1 12402.917,E2 12402.917} C_VEL
LIN {X 0,Y 490.7,Z 663.19,A -85,B 0,C 180,E1 12410.225,E2 12410.225} C_VEL
LIN {X 0,Y 490.69,Z 663.19,A -85,B 0,C 180,E1 12419.133,E2 12419.133} C_VEL
LIN {X 0,Y 490.379,Z 663.19,A -85,B 0,C 180,E1 12428.026,E2 12428.026} C_VEL
LIN {X 0,Y 489.954,Z 663.19,A -85,B 0,C 180,E1 12437.135,E2 12437.135} C_VEL
LIN {X 0,Y 489.757,Z 663.19,A -85,B 0,C 180,E1 12446.724,E2 12446.724} C_VEL
LIN {X 0,Y 490.198,Z 664.786,A -85,B 0,C 180,E1 12453.341,E2 12453.341} C_VEL
LIN {X 0,Y 528.797,Z 726.172,A -85,B 0,C 180,E1 12460.304,E2 12460.304} C_VEL
LIN {X 0,Y 546.899,Z 767.122,A -85,B 0,C 180,E1 12463.764,E2 12463.764} C_VEL
LIN {X 0,Y 536.037,Z 841.527,A -85,B 0,C 180,E1 12466.824,E2 12466.824} C_VEL
LIN {X 0,Y 522.464,Z 908.79,A -85,B 0,C 180,E1 12471.504,E2 12471.504} C_VEL
LIN {X 0,Y 509.514,Z 965.648,A -85,B 0,C 180,E1 12477.609,E2 12477.609} C_VEL
LIN {X 0,Y 499.357,Z 1011.894,A -85,B 0,C 180,E1 12485.081,E2 12485.081} C_VEL
LIN {X 0,Y 493.358,Z 1045.339,A -85,B 0,C 180,E1 12493.483,E2 12493.483} C_VEL
LIN {X 0,Y 491.219,Z 1064.445,A -85,B 0,C 180,E1 12502.015,E2 12502.015} C_VEL
LIN {X 0,Y 491.039,Z 1070.113,A -85,B 0,C 180,E1 12509.116,E2 12509.116} C_VEL
LIN {X 0,Y 491.512,Z 1065.666,A -85,B 0,C 180,E1 12517.089,E2 12517.089} C_VEL
LIN {X 0,Y 492.711,Z 1048.022,A -85,B 0,C 180,E1 12525.623,E2 12525.623} C_VEL
LIN {X 0,Y 497.336,Z 1018.863,A -85,B 0,C 180,E1 12533.504,E2 12533.504} C_VEL
LIN {X 0,Y 507.048,Z 975.858,A -85,B 0,C 180,E1 12541.057,E2 12541.057} C_VEL
LIN {X 0,Y 520.834,Z 918.724,A -85,B 0,C 180,E1 12547.717,E2 12547.717} C_VEL
LIN {X 0,Y 534.994,Z 854.7,A -85,B 0,C 180,E1 12552.57,E2 12552.57} C_VEL
LIN {X 0,Y 546.772,Z 783.487,A -85,B 0,C 180,E1 12555.896,E2 12555.896} C_VEL
LIN {X 0,Y 547.988,Z 762.907,A -85,B 0,C 180,E1 12556.691,E2 12556.691} C_VEL
LIN {X 0,Y 521.847,Z 712.248,A -85,B 0,C 180,E1 12561.737,E2 12561.737} C_VEL
LIN {X 0,Y 489.54,Z 663.19,A -85,B 0,C 180,E1 12568.767,E2 12568.767} C_VEL
LIN {X 0,Y 489.872,Z 663.19,A -85,B 0,C 180,E1 12579.106,E2 12579.106} C_VEL
LIN {X 0,Y 490.345,Z 663.19,A -85,B 0,C 180,E1 12588.373,E2 12588.373} C_VEL
LIN {X 0,Y 490.609,Z 663.19,A -85,B 0,C 180,E1 12597.321,E2 12597.321} C_VEL
LIN {X 0,Y 490.769,Z 663.19,A -85,B 0,C 180,E1 12604.415,E2 12604.415} C_VEL
LIN {X 0,Y 490.217,Z 663.19,A -85,B 0,C 180,E1 12613.408,E2 12613.408} C_VEL
LIN {X 0,Y 489.993,Z 663.19,A -85,B 0,C 180,E1 12622.759,E2 12622.759} C_VEL
LIN {X 0,Y 490.077,Z 664.769,A -85,B 0,C 180,E1 12628.764,E2 12628.764} C_VEL
LIN {X 0,Y 526.158,Z 718.694,A -85,B 0,C 180,E1 12636.167,E2 12636.167} C_VEL
LIN {X 0,Y 548.375,Z 766.324,A -85,B 0,C 180,E1 12640.784,E2 12640.784} C_VEL
LIN {X 0,Y 537.028,Z 837.575,A -85,B 0,C 180,E1 12643.846,E2 12643.846} C_VEL
LIN {X 0,Y 522.934,Z 903.471,A -85,B 0,C 180,E1 12648.584,E2 12648.584} C_VEL
LIN {X 0,Y 509.356,Z 959.982,A -85,B 0,C 180,E1 12654.879,E2 12654.879} C_VEL
LIN {X 0,Y 498.891,Z 1005.927,A -85,B 0,C 180,E1 12662.63,E2 12662.63} C_VEL
LIN {X 0,Y 493.058,Z 1038.262,A -85,B 0,C 180,E1 12671.159,E2 12671.159} C_VEL
LIN {X 0,Y 491.213,Z 1055.46,A -85,B 0,C 180,E1 12679.325,E2 12679.325} C_VEL
LIN {X 0,Y 491.271,Z 1060.57,A -85,B 0,C 180,E1 12687.773,E2 12687.773} C_VEL
LIN {X 0,Y 491.46,Z 1054.471,A -85,B 0,C 180,E1 12695.311,E2 12695.311} C_VEL
LIN {X 0,Y 493.049,Z 1036.555,A -85,B 0,C 180,E1 12703.336,E2 12703.336} C_VEL
LIN {X 0,Y 498.347,Z 1005.966,A -85,B 0,C 180,E1 12711.286,E2 12711.286} C_VEL
LIN {X 0,Y 508.625,Z 960.978,A -85,B 0,C 180,E1 12718.834,E2 12718.834} C_VEL
LIN {X 0,Y 522.286,Z 903.535,A -85,B 0,C 180,E1 12725.18,E2 12725.18} C_VEL
LIN {X 0,Y 535.777,Z 838.191,A -85,B 0,C 180,E1 12729.845,E2 12729.845} C_VEL
LIN {X 0,Y 546.428,Z 766.415,A -85,B 0,C 180,E1 12732.953,E2 12732.953} C_VEL
LIN {X 0,Y 519.216,Z 709.817,A -85,B 0,C 180,E1 12738.103,E2 12738.103} C_VEL
LIN {X 0,Y 489.645,Z 663.19,A -85,B 0,C 180,E1 12743.934,E2 12743.934} C_VEL
LIN {X 0,Y 481.633,Z 663.19,A -85,B 0,C 180,E1 12748.029,E2 12748.029} C_VEL
LIN {X 0,Y 481.939,Z 663.19,A -85,B 0,C 180,E1 12758.157,E2 12758.157} C_VEL
LIN {X 0,Y 482.897,Z 663.19,A -85,B 0,C 180,E1 12768.231,E2 12768.231} C_VEL
LIN {X 0,Y 482.69,Z 663.19,A -85,B 0,C 180,E1 12779.119,E2 12779.119} C_VEL
LIN {X 0,Y 482.381,Z 663.19,A -85,B 0,C 180,E1 12788.16,E2 12788.16} C_VEL
LIN {X 0,Y 481.93,Z 663.19,A -85,B 0,C 180,E1 12797.43,E2 12797.43} C_VEL
LIN {X 0,Y 481.78,Z 663.19,A -85,B 0,C 180,E1 12807.203,E2 12807.203} C_VEL
LIN {X 0,Y 482.189,Z 665.026,A -85,B 0,C 180,E1 12811.95,E2 12811.95} C_VEL
LIN {X 0,Y 519.483,Z 722.886,A -85,B 0,C 180,E1 12819.052,E2 12819.052} C_VEL
LIN {X 0,Y 540.916,Z 770.018,A -85,B 0,C 180,E1 12823.254,E2 12823.254} C_VEL
LIN {X 0,Y 529.732,Z 843.068,A -85,B 0,C 180,E1 12826.324,E2 12826.324} C_VEL
LIN {X 0,Y 515.763,Z 909.611,A -85,B 0,C 180,E1 12831.026,E2 12831.026} C_VEL
LIN {X 0,Y 502.088,Z 967.147,A -85,B 0,C 180,E1 12837.326,E2 12837.326} C_VEL
LIN {X 0,Y 491.576,Z 1012.862,A -85,B 0,C 180,E1 12844.903,E2 12844.903} C_VEL
LIN {X 0,Y 485.228,Z 1046.607,A -85,B 0,C 180,E1 12853.665,E2 12853.665} C_VEL
LIN {X 0,Y 483.258,Z 1064.367,A -85,B 0,C 180,E1 12861.883,E2 12861.883} C_VEL
LIN {X 0,Y 483.035,Z 1070.036,A -85,B 0,C 180,E1 12869.101,E2 12869.101} C_VEL
LIN {X 0,Y 483.518,Z 1065.587,A -85,B 0,C 180,E1 12877.207,E2 12877.207} C_VEL
LIN {X 0,Y 484.82,Z 1047.941,A -85,B 0,C 180,E1 12885.884,E2 12885.884} C_VEL
LIN {X 0,Y 490.045,Z 1017.443,A -85,B 0,C 180,E1 12894.183,E2 12894.183} C_VEL
LIN {X 0,Y 500.744,Z 972.684,A -85,B 0,C 180,E1 12902.003,E2 12902.003} C_VEL
LIN {X 0,Y 515.075,Z 915.764,A -85,B 0,C 180,E1 12908.573,E2 12908.573} C_VEL
LIN {X 0,Y 529.878,Z 850.914,A -85,B 0,C 180,E1 12913.411,E2 12913.411} C_VEL
LIN {X 0,Y 541.809,Z 780.379,A -85,B 0,C 180,E1 12916.619,E2 12916.619} C_VEL
LIN {X 0,Y 541.99,Z 765.592,A -85,B 0,C 180,E1 12917.271,E2 12917.271} C_VEL
LIN {X 0,Y 516.31,Z 715.49,A -85,B 0,C 180,E1 12922.469,E2 12922.469} C_VEL
LIN {X 0,Y 484.194,Z 669.119,A -85,B 0,C 180,E1 12929.41,E2 12929.41} C_VEL
LIN {X 0,Y 481.554,Z 663.19,A -85,B 0,C 180,E1 12930.401,E2 12930.401} C_VEL
LIN {X 0,Y 481.878,Z 663.19,A -85,B 0,C 180,E1 12940.667,E2 12940.667} C_VEL
LIN {X 0,Y 482.331,Z 663.19,A -85,B 0,C 180,E1 12950.014,E2 12950.014} C_VEL
LIN {X 0,Y 482.455,Z 663.19,A -85,B 0,C 180,E1 12959.079,E2 12959.079} C_VEL
LIN {X 0,Y 482.373,Z 663.19,A -85,B 0,C 180,E1 12966.303,E2 12966.303} C_VEL
LIN {X 0,Y 482.127,Z 663.19,A -85,B 0,C 180,E1 12976.401,E2 12976.401} C_VEL
LIN {X 0,Y 481.956,Z 663.19,A -85,B 0,C 180,E1 12986.66,E2 12986.66} C_VEL
LIN {X 0,Y 513.495,Z 710.42,A -85,B 0,C 180,E1 12994.08,E2 12994.08} C_VEL
LIN {X 0,Y 540.939,Z 763.77,A -85,B 0,C 180,E1 12999.8,E2 12999.8} C_VEL
LIN {X 0,Y 541.871,Z 775.231,A -85,B 0,C 180,E1 13000.447,E2 13000.447} C_VEL
LIN {X 0,Y 529.815,Z 845.039,A -85,B 0,C 180,E1 13003.668,E2 13003.668} C_VEL
LIN {X 0,Y 514.88,Z 910.279,A -85,B 0,C 180,E1 13008.637,E2 13008.637} C_VEL
LIN {X 0,Y 500.772,Z 966.275,A -85,B 0,C 180,E1 13015.248,E2 13015.248} C_VEL
LIN {X 0,Y 490.175,Z 1011.275,A -85,B 0,C 180,E1 13023.347,E2 13023.347} C_VEL
LIN {X 0,Y 484.554,Z 1041.985,A -85,B 0,C 180,E1 13032.234,E2 13032.234} C_VEL
LIN {X 0,Y 483.214,Z 1056.682,A -85,B 0,C 180,E1 13040.061,E2 13040.061} C_VEL
LIN {X 0,Y 483.275,Z 1060.4,A -85,B 0,C 180,E1 13049.101,E2 13049.101} C_VEL
LIN {X 0,Y 483.357,Z 1053.216,A -85,B 0,C 180,E1 13056.304,E2 13056.304} C_VEL
LIN {X 0,Y 485.477,Z 1035.09,A -85,B 0,C 180,E1 13064.141,E2 13064.141} C_VEL
LIN {X 0,Y 492.077,Z 1001.301,A -85,B 0,C 180,E1 13072.656,E2 13072.656} C_VEL
LIN {X 0,Y 503.502,Z 953.386,A -85,B 0,C 180,E1 13080.339,E2 13080.339} C_VEL
LIN {X 0,Y 517.82,Z 894.617,A -85,B 0,C 180,E1 13086.505,E2 13086.505} C_VEL
LIN {X 0,Y 531.481,Z 828.954,A -85,B 0,C 180,E1 13090.94,E2 13090.94} C_VEL
LIN {X 0,Y 539.534,Z 765.223,A -85,B 0,C 180,E1 13093.743,E2 13093.743} C_VEL
LIN {X 0,Y 508.386,Z 704.626,A -85,B 0,C 180,E1 13099.716,E2 13099.716} C_VEL
LIN {X 0,Y 481.626,Z 663.19,A -85,B 0,C 180,E1 13105.239,E2 13105.239} C_VEL
LIN {X 0,Y 481.633,Z 663.19,A -85,B 0,C 180,E1 13108.029,E2 13108.029} C_VEL
LIN {X 0,Y 473.75,Z 663.19,A -85,B 0,C 180,E1 13112.191,E2 13112.191} C_VEL
LIN {X 0,Y 474.169,Z 663.19,A -85,B 0,C 180,E1 13122.318,E2 13122.318} C_VEL
LIN {X 0,Y 474.708,Z 663.19,A -85,B 0,C 180,E1 13129.892,E2 13129.892} C_VEL
LIN {X 0,Y 474.704,Z 663.19,A -85,B 0,C 180,E1 13139.104,E2 13139.104} C_VEL
LIN {X 0,Y 474.359,Z 663.19,A -85,B 0,C 180,E1 13148.299,E2 13148.299} C_VEL
LIN {X 0,Y 473.886,Z 663.19,A -85,B 0,C 180,E1 13157.735,E2 13157.735} C_VEL
LIN {X 0,Y 473.762,Z 663.19,A -85,B 0,C 180,E1 13168.332,E2 13168.332} C_VEL
LIN {X 0,Y 474.183,Z 665.293,A -85,B 0,C 180,E1 13170.458,E2 13170.458} C_VEL
LIN {X 0,Y 508.999,Z 717.647,A -85,B 0,C 180,E1 13177.508,E2 13177.508} C_VEL
LIN {X 0,Y 535.031,Z 772.375,A -85,B 0,C 180,E1 13182.715,E2 13182.715} C_VEL
LIN {X 0,Y 523.47,Z 844.578,A -85,B 0,C 180,E1 13185.809,E2 13185.809} C_VEL
LIN {X 0,Y 508.856,Z 911.519,A -85,B 0,C 180,E1 13190.631,E2 13190.631} C_VEL
LIN {X 0,Y 494.64,Z 968.569,A -85,B 0,C 180,E1 13197.033,E2 13197.033} C_VEL
LIN {X 0,Y 483.561,Z 1014.917,A -85,B 0,C 180,E1 13204.954,E2 13204.954} C_VEL
LIN {X 0,Y 477.117,Z 1047.869,A -85,B 0,C 180,E1 13213.854,E2 13213.854} C_VEL
LIN {X 0,Y 475.294,Z 1064.289,A -85,B 0,C 180,E1 13221.746,E2 13221.746} C_VEL
LIN {X 0,Y 475.043,Z 1069.958,A -85,B 0,C 180,E1 13229.086,E2 13229.086} C_VEL
LIN {X 0,Y 475.516,Z 1065.508,A -85,B 0,C 180,E1 13237.329,E2 13237.329} C_VEL
LIN {X 0,Y 476.766,Z 1049.213,A -85,B 0,C 180,E1 13245.686,E2 13245.686} C_VEL
LIN {X 0,Y 481.906,Z 1020.186,A -85,B 0,C 180,E1 13253.981,E2 13253.981} C_VEL
LIN {X 0,Y 492.725,Z 976.59,A -85,B 0,C 180,E1 13261.956,E2 13261.956} C_VEL
LIN {X 0,Y 507.699,Z 919.766,A -85,B 0,C 180,E1 13268.773,E2 13268.773} C_VEL
LIN {X 0,Y 522.962,Z 856.081,A -85,B 0,C 180,E1 13273.711,E2 13273.711} C_VEL
LIN {X 0,Y 535.463,Z 786.106,A -85,B 0,C 180,E1 13277.062,E2 13277.062} C_VEL
LIN {X 0,Y 536.261,Z 769.006,A -85,B 0,C 180,E1 13277.803,E2 13277.803} C_VEL
LIN {X 0,Y 511.129,Z 719.141,A -85,B 0,C 180,E1 13283.164,E2 13283.164} C_VEL
LIN {X 0,Y 480.095,Z 674.285,A -85,B 0,C 180,E1 13290.135,E2 13290.135} C_VEL
LIN {X 0,Y 473.549,Z 663.19,A -85,B 0,C 180,E1 13292.284,E2 13292.284} C_VEL
LIN {X 0,Y 473.888,Z 663.19,A -85,B 0,C 180,E1 13302.265,E2 13302.265} C_VEL
LIN {X 0,Y 474.366,Z 663.19,A -85,B 0,C 180,E1 13311.702,E2 13311.702} C_VEL
LIN {X 0,Y 474.681,Z 663.19,A -85,B 0,C 180,E1 13320.896,E2 13320.896} C_VEL
LIN {X 0,Y 474.403,Z 663.19,A -85,B 0,C 180,E1 13330.115,E2 13330.115} C_VEL
LIN {X 0,Y 474.129,Z 663.19,A -85,B 0,C 180,E1 13339.62,E2 13339.62} C_VEL
LIN {X 0,Y 474.139,Z 665.06,A -85,B 0,C 180,E1 13345.306,E2 13345.306} C_VEL
LIN {X 0,Y 506.772,Z 711.675,A -85,B 0,C 180,E1 13353.047,E2 13353.047} C_VEL
LIN {X 0,Y 533.429,Z 762.894,A -85,B 0,C 180,E1 13358.838,E2 13358.838} C_VEL
LIN {X 0,Y 536.436,Z 775.63,A -85,B 0,C 180,E1 13359.822,E2 13359.822} C_VEL
LIN {X 0,Y 523.899,Z 845.686,A -85,B 0,C 180,E1 13363.079,E2 13363.079} C_VEL
LIN {X 0,Y 508.328,Z 911.184,A -85,B 0,C 180,E1 13368.128,E2 13368.128} C_VEL
LIN {X 0,Y 493.557,Z 967.247,A -85,B 0,C 180,E1 13374.856,E2 13374.856} C_VEL
LIN {X 0,Y 482.744,Z 1011.17,A -85,B 0,C 180,E1 13382.904,E2 13382.904} C_VEL
LIN {X 0,Y 476.689,Z 1041.937,A -85,B 0,C 180,E1 13391.931,E2 13391.931} C_VEL
LIN {X 0,Y 475.214,Z 1056.692,A -85,B 0,C 180,E1 13399.891,E2 13399.891} C_VEL
LIN {X 0,Y 475.288,Z 1060.487,A -85,B 0,C 180,E1 13409.086,E2 13409.086} C_VEL
LIN {X 0,Y 475.401,Z 1053.38,A -85,B 0,C 180,E1 13416.41,E2 13416.41} C_VEL
LIN {X 0,Y 477.963,Z 1033.807,A -85,B 0,C 180,E1 13424.875,E2 13424.875} C_VEL
LIN {X 0,Y 485.176,Z 999.214,A -85,B 0,C 180,E1 13433.484,E2 13433.484} C_VEL
LIN {X 0,Y 497.213,Z 951.075,A -85,B 0,C 180,E1 13441.157,E2 13441.157} C_VEL
LIN {X 0,Y 511.956,Z 892.598,A -85,B 0,C 180,E1 13447.256,E2 13447.256} C_VEL
LIN {X 0,Y 526.285,Z 825.418,A -85,B 0,C 180,E1 13451.735,E2 13451.735} C_VEL
LIN {X 0,Y 533.413,Z 768.142,A -85,B 0,C 180,E1 13454.291,E2 13454.291} C_VEL
LIN {X 0,Y 503.605,Z 709.159,A -85,B 0,C 180,E1 13460.283,E2 13460.283} C_VEL
LIN {X 0,Y 473.638,Z 663.19,A -85,B 0,C 180,E1 13466.742,E2 13466.742} C_VEL
LIN {X 0,Y 473.75,Z 663.19,A -85,B 0,C 180,E1 13472.191,E2 13472.191} C_VEL
LIN {X 0,Y 465.825,Z 663.19,A -85,B 0,C 180,E1 13476.406,E2 13476.406} C_VEL
LIN {X 0,Y 466.671,Z 663.19,A -85,B 0,C 180,E1 13485.902,E2 13485.902} C_VEL
LIN {X 0,Y 467.078,Z 663.19,A -85,B 0,C 180,E1 13497.226,E2 13497.226} C_VEL
LIN {X 0,Y 466.429,Z 663.19,A -85,B 0,C 180,E1 13507.44,E2 13507.44} C_VEL
LIN {X 0,Y 465.951,Z 663.19,A -85,B 0,C 180,E1 13516.249,E2 13516.249} C_VEL
LIN {X 0,Y 465.645,Z 663.19,A -85,B 0,C 180,E1 13526.42,E2 13526.42} C_VEL
LIN {X 0,Y 466.036,Z 665.144,A -85,B 0,C 180,E1 13528.805,E2 13528.805} C_VEL
LIN {X 0,Y 499.681,Z 714.637,A -85,B 0,C 180,E1 13536.08,E2 13536.08} C_VEL
LIN {X 0,Y 529.213,Z 773.73,A -85,B 0,C 180,E1 13542.122,E2 13542.122} C_VEL
LIN {X 0,Y 517.125,Z 846.833,A -85,B 0,C 180,E1 13545.327,E2 13545.327} C_VEL
LIN {X 0,Y 501.9,Z 913.439,A -85,B 0,C 180,E1 13550.235,E2 13550.235} C_VEL
LIN {X 0,Y 487.205,Z 970.034,A -85,B 0,C 180,E1 13556.739,E2 13556.739} C_VEL
LIN {X 0,Y 475.662,Z 1016.315,A -85,B 0,C 180,E1 13564.864,E2 13564.864} C_VEL
LIN {X 0,Y 469.254,Z 1047.881,A -85,B 0,C 180,E1 13573.616,E2 13573.616} C_VEL
LIN {X 0,Y 467.233,Z 1065.2,A -85,B 0,C 180,E1 13582.364,E2 13582.364} C_VEL
LIN {X 0,Y 467.524,Z 1069.884,A -85,B 0,C 180,E1 13590.93,E2 13590.93} C_VEL
LIN {X 0,Y 467.399,Z 1062.898,A -85,B 0,C 180,E1 13599.336,E2 13599.336} C_VEL
LIN {X 0,Y 469.785,Z 1043.777,A -85,B 0,C 180,E1 13607.858,E2 13607.858} C_VEL
LIN {X 0,Y 477.498,Z 1008.532,A -85,B 0,C 180,E1 13616.881,E2 13616.881} C_VEL
LIN {X 0,Y 490.248,Z 960.536,A -85,B 0,C 180,E1 13624.728,E2 13624.728} C_VEL
LIN {X 0,Y 505.842,Z 902.533,A -85,B 0,C 180,E1 13630.956,E2 13630.956} C_VEL
LIN {X 0,Y 521.599,Z 835.114,A -85,B 0,C 180,E1 13635.556,E2 13635.556} C_VEL
LIN {X 0,Y 530.769,Z 772.781,A -85,B 0,C 180,E1 13638.305,E2 13638.305} C_VEL
LIN {X 0,Y 505.889,Z 722.722,A -85,B 0,C 180,E1 13643.897,E2 13643.897} C_VEL
LIN {X 0,Y 474.675,Z 677.041,A -85,B 0,C 180,E1 13651.272,E2 13651.272} C_VEL
LIN {X 0,Y 465.597,Z 663.19,A -85,B 0,C 180,E1 13654.257,E2 13654.257} C_VEL
LIN {X 0,Y 465.98,Z 663.19,A -85,B 0,C 180,E1 13663.906,E2 13663.906} C_VEL
LIN {X 0,Y 466.591,Z 663.19,A -85,B 0,C 180,E1 13673.442,E2 13673.442} C_VEL
LIN {X 0,Y 467.078,Z 663.19,A -85,B 0,C 180,E1 13682.774,E2 13682.774} C_VEL
LIN {X 0,Y 466.299,Z 663.19,A -85,B 0,C 180,E1 13692.194,E2 13692.194} C_VEL
LIN {X 0,Y 465.971,Z 663.19,A -85,B 0,C 180,E1 13701.977,E2 13701.977} C_VEL
LIN {X 0,Y 466.27,Z 665.595,A -85,B 0,C 180,E1 13703.351,E2 13703.351} C_VEL
LIN {X 0,Y 495.208,Z 705.374,A -85,B 0,C 180,E1 13710.867,E2 13710.867} C_VEL
LIN {X 0,Y 523.231,Z 755.703,A -85,B 0,C 180,E1 13717.155,E2 13717.155} C_VEL
LIN {X 0,Y 530.693,Z 778.486,A -85,B 0,C 180,E1 13719.275,E2 13719.275} C_VEL
LIN {X 0,Y 517.628,Z 848.181,A -85,B 0,C 180,E1 13722.592,E2 13722.592} C_VEL
LIN {X 0,Y 501.603,Z 912.8,A -85,B 0,C 180,E1 13727.672,E2 13727.672} C_VEL
LIN {X 0,Y 486.194,Z 968.873,A -85,B 0,C 180,E1 13734.548,E2 13734.548} C_VEL
LIN {X 0,Y 474.993,Z 1012.144,A -85,B 0,C 180,E1 13742.698,E2 13742.698} C_VEL
LIN {X 0,Y 468.854,Z 1041.903,A -85,B 0,C 180,E1 13751.618,E2 13751.618} C_VEL
LIN {X 0,Y 467.23,Z 1056.703,A -85,B 0,C 180,E1 13759.717,E2 13759.717} C_VEL
LIN {X 0,Y 467.287,Z 1060.574,A -85,B 0,C 180,E1 13769.07,E2 13769.07} C_VEL
LIN {X 0,Y 467.417,Z 1053.545,A -85,B 0,C 180,E1 13776.519,E2 13776.519} C_VEL
LIN {X 0,Y 470.211,Z 1033.709,A -85,B 0,C 180,E1 13785.226,E2 13785.226} C_VEL
LIN {X 0,Y 478.003,Z 998.305,A -85,B 0,C 180,E1 13794.107,E2 13794.107} C_VEL
LIN {X 0,Y 490.808,Z 949.616,A -85,B 0,C 180,E1 13801.881,E2 13801.881} C_VEL
LIN {X 0,Y 506.336,Z 889.899,A -85,B 0,C 180,E1 13808.083,E2 13808.083} C_VEL
LIN {X 0,Y 520.993,Z 822.388,A -85,B 0,C 180,E1 13812.505,E2 13812.505} C_VEL
LIN {X 0,Y 527.484,Z 771.388,A -85,B 0,C 180,E1 13814.821,E2 13814.821} C_VEL
LIN {X 0,Y 498.654,Z 713.237,A -85,B 0,C 180,E1 13820.907,E2 13820.907} C_VEL
LIN {X 0,Y 465.645,Z 663.19,A -85,B 0,C 180,E1 13828.316,E2 13828.316} C_VEL
LIN {X 0,Y 465.825,Z 663.19,A -85,B 0,C 180,E1 13836.406,E2 13836.406} C_VEL
LIN {X 0,Y 457.992,Z 663.19,A -85,B 0,C 180,E1 13840.693,E2 13840.693} C_VEL
LIN {X 0,Y 458.72,Z 663.19,A -85,B 0,C 180,E1 13849.536,E2 13849.536} C_VEL
LIN {X 0,Y 458.706,Z 663.19,A -85,B 0,C 180,E1 13859.073,E2 13859.073} C_VEL
LIN {X 0,Y 458.323,Z 663.19,A -85,B 0,C 180,E1 13868.591,E2 13868.591} C_VEL
LIN {X 0,Y 457.808,Z 663.19,A -85,B 0,C 180,E1 13878.38,E2 13878.38} C_VEL
LIN {X 0,Y 457.87,Z 665.029,A -85,B 0,C 180,E1 13887.001,E2 13887.001} C_VEL
LIN {X 0,Y 489.496,Z 710.404,A -85,B 0,C 180,E1 13894.372,E2 13894.372} C_VEL
LIN {X 0,Y 518.418,Z 765.667,A -85,B 0,C 180,E1 13900.466,E2 13900.466} C_VEL
LIN {X 0,Y 522.963,Z 780.867,A -85,B 0,C 180,E1 13901.728,E2 13901.728} C_VEL
LIN {X 0,Y 509.795,Z 853.719,A -85,B 0,C 180,E1 13905.119,E2 13905.119} C_VEL
LIN {X 0,Y 493.894,Z 919.29,A -85,B 0,C 180,E1 13910.214,E2 13910.214} C_VEL
LIN {X 0,Y 478.852,Z 974.97,A -85,B 0,C 180,E1 13916.945,E2 13916.945} C_VEL
LIN {X 0,Y 467.524,Z 1018.743,A -85,B 0,C 180,E1 13925,E2 13925} C_VEL
LIN {X 0,Y 460.887,Z 1050.217,A -85,B 0,C 180,E1 13934.25,E2 13934.25} C_VEL
LIN {X 0,Y 459.242,Z 1065.116,A -85,B 0,C 180,E1 13942.23,E2 13942.23} C_VEL
LIN {X 0,Y 459.512,Z 1069.806,A -85,B 0,C 180,E1 13950.946,E2 13950.946} C_VEL
LIN {X 0,Y 459.439,Z 1062.83,A -85,B 0,C 180,E1 13959.499,E2 13959.499} C_VEL
LIN {X 0,Y 462.346,Z 1042.284,A -85,B 0,C 180,E1 13968.65,E2 13968.65} C_VEL
LIN {X 0,Y 470.855,Z 1006.007,A -85,B 0,C 180,E1 13977.839,E2 13977.839} C_VEL
LIN {X 0,Y 484.345,Z 957.69,A -85,B 0,C 180,E1 13985.671,E2 13985.671} C_VEL
LIN {X 0,Y 500.772,Z 898.904,A -85,B 0,C 180,E1 13991.896,E2 13991.896} C_VEL
LIN {X 0,Y 516.771,Z 831.54,A -85,B 0,C 180,E1 13996.402,E2 13996.402} C_VEL
LIN {X 0,Y 525.144,Z 776.065,A -85,B 0,C 180,E1 13998.865,E2 13998.865} C_VEL
LIN {X 0,Y 500.394,Z 725.737,A -85,B 0,C 180,E1 14004.719,E2 14004.719} C_VEL
LIN {X 0,Y 470.883,Z 682.82,A -85,B 0,C 180,E1 14011.983,E2 14011.983} C_VEL
LIN {X 0,Y 457.585,Z 663.19,A -85,B 0,C 180,E1 14016.522,E2 14016.522} C_VEL
LIN {X 0,Y 458.278,Z 663.19,A -85,B 0,C 180,E1 14027.46,E2 14027.46} C_VEL
LIN {X 0,Y 458.629,Z 663.19,A -85,B 0,C 180,E1 14037.134,E2 14037.134} C_VEL
LIN {X 0,Y 458.685,Z 663.19,A -85,B 0,C 180,E1 14044.725,E2 14044.725} C_VEL
LIN {X 0,Y 458.083,Z 663.19,A -85,B 0,C 180,E1 14054.368,E2 14054.368} C_VEL
LIN {X 0,Y 458.173,Z 665.021,A -85,B 0,C 180,E1 14061.051,E2 14061.051} C_VEL
LIN {X 0,Y 487.304,Z 704.714,A -85,B 0,C 180,E1 14069.355,E2 14069.355} C_VEL
LIN {X 0,Y 515.2,Z 753.691,A -85,B 0,C 180,E1 14075.943,E2 14075.943} C_VEL
LIN {X 0,Y 524.965,Z 781.451,A -85,B 0,C 180,E1 14078.718,E2 14078.718} C_VEL
LIN {X 0,Y 511.484,Z 850.31,A -85,B 0,C 180,E1 14082.071,E2 14082.071} C_VEL
LIN {X 0,Y 494.793,Z 914.86,A -85,B 0,C 180,E1 14087.248,E2 14087.248} C_VEL
LIN {X 0,Y 479.01,Z 969.956,A -85,B 0,C 180,E1 14094.15,E2 14094.15} C_VEL
LIN {X 0,Y 467.369,Z 1012.784,A -85,B 0,C 180,E1 14102.406,E2 14102.406} C_VEL
LIN {X 0,Y 460.787,Z 1043.031,A -85,B 0,C 180,E1 14111.781,E2 14111.781} C_VEL
LIN {X 0,Y 459.245,Z 1056.72,A -85,B 0,C 180,E1 14119.536,E2 14119.536} C_VEL
LIN {X 0,Y 459.217,Z 1060.898,A -85,B 0,C 180,E1 14127.745,E2 14127.745} C_VEL
LIN {X 0,Y 459.463,Z 1055.045,A -85,B 0,C 180,E1 14135.682,E2 14135.682} C_VEL
LIN {X 0,Y 461.624,Z 1037.403,A -85,B 0,C 180,E1 14144.262,E2 14144.262} C_VEL
LIN {X 0,Y 468.58,Z 1005.669,A -85,B 0,C 180,E1 14153.029,E2 14153.029} C_VEL
LIN {X 0,Y 481.052,Z 959.781,A -85,B 0,C 180,E1 14161.076,E2 14161.076} C_VEL
LIN {X 0,Y 497,Z 901.934,A -85,B 0,C 180,E1 14167.637,E2 14167.637} C_VEL
LIN {X 0,Y 512.34,Z 837.006,A -85,B 0,C 180,E1 14172.346,E2 14172.346} C_VEL
LIN {X 0,Y 521.703,Z 775.05,A -85,B 0,C 180,E1 14175.321,E2 14175.321} C_VEL
LIN {X 0,Y 493.972,Z 718.02,A -85,B 0,C 180,E1 14181.491,E2 14181.491} C_VEL
LIN {X 0,Y 461.113,Z 669.808,A -85,B 0,C 180,E1 14188.935,E2 14188.935} C_VEL
LIN {X 0,Y 457.637,Z 663.19,A -85,B 0,C 180,E1 14190.214,E2 14190.214} C_VEL
LIN {X 0,Y 457.992,Z 663.19,A -85,B 0,C 180,E1 14200.693,E2 14200.693} C_VEL
LIN {X 0,Y 450.469,Z 663.19,A -85,B 0,C 180,E1 14205.088,E2 14205.088} C_VEL
LIN {X 0,Y 450.662,Z 663.19,A -85,B 0,C 180,E1 14215.191,E2 14215.191} C_VEL
LIN {X 0,Y 450.83,Z 663.19,A -85,B 0,C 180,E1 14224.849,E2 14224.849} C_VEL
LIN {X 0,Y 450.044,Z 663.19,A -85,B 0,C 180,E1 14234.673,E2 14234.673} C_VEL
LIN {X 0,Y 449.758,Z 664.795,A -85,B 0,C 180,E1 14245.023,E2 14245.023} C_VEL
LIN {X 0,Y 481.647,Z 709.679,A -85,B 0,C 180,E1 14253.033,E2 14253.033} C_VEL
LIN {X 0,Y 510.192,Z 763.224,A -85,B 0,C 180,E1 14259.303,E2 14259.303} C_VEL
LIN {X 0,Y 517.003,Z 784.21,A -85,B 0,C 180,E1 14261.203,E2 14261.203} C_VEL
LIN {X 0,Y 503.514,Z 855.495,A -85,B 0,C 180,E1 14264.595,E2 14264.595} C_VEL
LIN {X 0,Y 486.864,Z 921.458,A -85,B 0,C 180,E1 14269.829,E2 14269.829} C_VEL
LIN {X 0,Y 471.175,Z 977.231,A -85,B 0,C 180,E1 14276.757,E2 14276.757} C_VEL
LIN {X 0,Y 459.387,Z 1020.907,A -85,B 0,C 180,E1 14285.112,E2 14285.112} C_VEL
LIN {X 0,Y 452.802,Z 1051.266,A -85,B 0,C 180,E1 14294.46,E2 14294.46} C_VEL
LIN {X 0,Y 451.274,Z 1066.366,A -85,B 0,C 180,E1 14303.246,E2 14303.246} C_VEL
LIN {X 0,Y 451.501,Z 1069.73,A -85,B 0,C 180,E1 14310.963,E2 14310.963} C_VEL
LIN {X 0,Y 451.475,Z 1062.768,A -85,B 0,C 180,E1 14319.669,E2 14319.669} C_VEL
LIN {X 0,Y 454.596,Z 1042.252,A -85,B 0,C 180,E1 14328.98,E2 14328.98} C_VEL
LIN {X 0,Y 463.564,Z 1006.018,A -85,B 0,C 180,E1 14338.316,E2 14338.316} C_VEL
LIN {X 0,Y 477.665,Z 957.757,A -85,B 0,C 180,E1 14346.248,E2 14346.248} C_VEL
LIN {X 0,Y 494.714,Z 899.047,A -85,B 0,C 180,E1 14352.529,E2 14352.529} C_VEL
LIN {X 0,Y 511.275,Z 831.836,A -85,B 0,C 180,E1 14357.053,E2 14357.053} C_VEL
LIN {X 0,Y 519.539,Z 779.498,A -85,B 0,C 180,E1 14359.434,E2 14359.434} C_VEL
LIN {X 0,Y 495.182,Z 729.354,A -85,B 0,C 180,E1 14365.476,E2 14365.476} C_VEL
LIN {X 0,Y 465.429,Z 685.056,A -85,B 0,C 180,E1 14373.271,E2 14373.271} C_VEL
LIN {X 0,Y 449.67,Z 663.19,A -85,B 0,C 180,E1 14379.22,E2 14379.22} C_VEL
LIN {X 0,Y 450.283,Z 663.19,A -85,B 0,C 180,E1 14389.295,E2 14389.295} C_VEL
LIN {X 0,Y 450.466,Z 663.19,A -85,B 0,C 180,E1 14399.014,E2 14399.014} C_VEL
LIN {X 0,Y 450.343,Z 663.19,A -85,B 0,C 180,E1 14406.753,E2 14406.753} C_VEL
LIN {X 0,Y 450.058,Z 663.19,A -85,B 0,C 180,E1 14416.636,E2 14416.636} C_VEL
LIN {X 0,Y 450.316,Z 665.249,A -85,B 0,C 180,E1 14418.525,E2 14418.525} C_VEL
LIN {X 0,Y 475.582,Z 698.488,A -85,B 0,C 180,E1 14426.708,E2 14426.708} C_VEL
LIN {X 0,Y 503.903,Z 745.185,A -85,B 0,C 180,E1 14433.842,E2 14433.842} C_VEL
LIN {X 0,Y 519.362,Z 784.057,A -85,B 0,C 180,E1 14438.137,E2 14438.137} C_VEL
LIN {X 0,Y 505.139,Z 853.434,A -85,B 0,C 180,E1 14441.598,E2 14441.598} C_VEL
LIN {X 0,Y 487.826,Z 917.566,A -85,B 0,C 180,E1 14446.875,E2 14446.875} C_VEL
LIN {X 0,Y 471.732,Z 971.333,A -85,B 0,C 180,E1 14453.794,E2 14453.794} C_VEL
LIN {X 0,Y 459.853,Z 1012.912,A -85,B 0,C 180,E1 14461.971,E2 14461.971} C_VEL
LIN {X 0,Y 452.997,Z 1043.013,A -85,B 0,C 180,E1 14471.457,E2 14471.457} C_VEL
LIN {X 0,Y 451.261,Z 1056.743,A -85,B 0,C 180,E1 14479.349,E2 14479.349} C_VEL
LIN {X 0,Y 451.2,Z 1060.978,A -85,B 0,C 180,E1 14487.742,E2 14487.742} C_VEL
LIN {X 0,Y 451.482,Z 1055.178,A -85,B 0,C 180,E1 14495.783,E2 14495.783} C_VEL
LIN {X 0,Y 453.768,Z 1037.594,A -85,B 0,C 180,E1 14504.515,E2 14504.515} C_VEL
LIN {X 0,Y 461.223,Z 1005.508,A -85,B 0,C 180,E1 14513.516,E2 14513.516} C_VEL
LIN {X 0,Y 474.088,Z 960.096,A -85,B 0,C 180,E1 14521.585,E2 14521.585} C_VEL
LIN {X 0,Y 490.62,Z 902.427,A -85,B 0,C 180,E1 14528.207,E2 14528.207} C_VEL
LIN {X 0,Y 506.374,Z 837.884,A -85,B 0,C 180,E1 14532.942,E2 14532.942} C_VEL
LIN {X 0,Y 516.201,Z 779.599,A -85,B 0,C 180,E1 14535.733,E2 14535.733} C_VEL
LIN {X 0,Y 489.682,Z 723.469,A -85,B 0,C 180,E1 14541.982,E2 14541.982} C_VEL
LIN {X 0,Y 458.303,Z 676.732,A -85,B 0,C 180,E1 14549.346,E2 14549.346} C_VEL
LIN {X 0,Y 449.657,Z 663.19,A -85,B 0,C 180,E1 14551.924,E2 14551.924} C_VEL
LIN {X 0,Y 450.034,Z 663.19,A -85,B 0,C 180,E1 14561.335,E2 14561.335} C_VEL
LIN {X 0,Y 450.469,Z 663.19,A -85,B 0,C 180,E1 14565.088,E2 14565.088} C_VEL
LIN {X 0,Y 442.609,Z 663.19,A -85,B 0,C 180,E1 14569.547,E2 14569.547} C_VEL
LIN {X 0,Y 442.731,Z 663.19,A -85,B 0,C 180,E1 14579.039,E2 14579.039} C_VEL
LIN {X 0,Y 442.295,Z 663.19,A -85,B 0,C 180,E1 14588.905,E2 14588.905} C_VEL
LIN {X 0,Y 441.72,Z 663.19,A -85,B 0,C 180,E1 14599.255,E2 14599.255} C_VEL
LIN {X 0,Y 441.834,Z 664.956,A -85,B 0,C 180,E1 14602.887,E2 14602.887} C_VEL
LIN {X 0,Y 472.004,Z 706.521,A -85,B 0,C 180,E1 14611.189,E2 14611.189} C_VEL
LIN {X 0,Y 500.382,Z 757.24,A -85,B 0,C 180,E1 14617.714,E2 14617.714} C_VEL
LIN {X 0,Y 511.258,Z 786.253,A -85,B 0,C 180,E1 14620.614,E2 14620.614} C_VEL
LIN {X 0,Y 497.161,Z 857.878,A -85,B 0,C 180,E1 14624.1,E2 14624.1} C_VEL
LIN {X 0,Y 480.001,Z 923.144,A -85,B 0,C 180,E1 14629.386,E2 14629.386} C_VEL
LIN {X 0,Y 463.653,Z 978.877,A -85,B 0,C 180,E1 14636.481,E2 14636.481} C_VEL
LIN {X 0,Y 451.305,Z 1022.722,A -85,B 0,C 180,E1 14645.165,E2 14645.165} C_VEL
LIN {X 0,Y 444.929,Z 1051.151,A -85,B 0,C 180,E1 14654.178,E2 14654.178} C_VEL
LIN {X 0,Y 443.27,Z 1066.276,A -85,B 0,C 180,E1 14663.124,E2 14663.124} C_VEL
LIN {X 0,Y 443.502,Z 1069.654,A -85,B 0,C 180,E1 14670.98,E2 14670.98} C_VEL
LIN {X 0,Y 443.509,Z 1062.711,A -85,B 0,C 180,E1 14679.844,E2 14679.844} C_VEL
LIN {X 0,Y 446.88,Z 1042.225,A -85,B 0,C 180,E1 14689.321,E2 14689.321} C_VEL
LIN {X 0,Y 456.267,Z 1006.033,A -85,B 0,C 180,E1 14698.811,E2 14698.811} C_VEL
LIN {X 0,Y 470.997,Z 957.903,A -85,B 0,C 180,E1 14706.833,E2 14706.833} C_VEL
LIN {X 0,Y 488.865,Z 898.659,A -85,B 0,C 180,E1 14713.225,E2 14713.225} C_VEL
LIN {X 0,Y 506.076,Z 830.816,A -85,B 0,C 180,E1 14717.79,E2 14717.79} C_VEL
LIN {X 0,Y 513.906,Z 782.88,A -85,B 0,C 180,E1 14720.007,E2 14720.007} C_VEL
LIN {X 0,Y 490.01,Z 732.985,A -85,B 0,C 180,E1 14726.255,E2 14726.255} C_VEL
LIN {X 0,Y 462.472,Z 691.787,A -85,B 0,C 180,E1 14733.809,E2 14733.809} C_VEL
LIN {X 0,Y 444.85,Z 669.585,A -85,B 0,C 180,E1 14740.374,E2 14740.374} C_VEL
LIN {X 0,Y 441.786,Z 663.19,A -85,B 0,C 180,E1 14742.483,E2 14742.483} C_VEL
LIN {X 0,Y 442.555,Z 663.19,A -85,B 0,C 180,E1 14753.084,E2 14753.084} C_VEL
LIN {X 0,Y 443.014,Z 663.19,A -85,B 0,C 180,E1 14762.924,E2 14762.924} C_VEL
LIN {X 0,Y 442.187,Z 663.19,A -85,B 0,C 180,E1 14772.87,E2 14772.87} C_VEL
LIN {X 0,Y 442.283,Z 665.215,A -85,B 0,C 180,E1 14775.447,E2 14775.447} C_VEL
LIN {X 0,Y 459.808,Z 687.978,A -85,B 0,C 180,E1 14782.415,E2 14782.415} C_VEL
LIN {X 0,Y 486.276,Z 726.446,A -85,B 0,C 180,E1 14789.938,E2 14789.938} C_VEL
LIN {X 0,Y 509.963,Z 774.173,A -85,B 0,C 180,E1 14796.243,E2 14796.243} C_VEL
LIN {X 0,Y 513.467,Z 788.839,A -85,B 0,C 180,E1 14797.625,E2 14797.625} C_VEL
